// NETWORK 5
//   TCP_clear_error: <<<<<<<<<<<<<<<<<<<<<<<<<<<<<clear error>>>>>>>>>>>>>>>>>>>>>>>>>>>>>>>>>
//   axisdata[1].Axis_Error: A-0-0021.09 -RD- Axis reports error
//   axisdata[2].Axis_Error: A-0-0021.09 -RD- Axis reports error
//   axisdata[3].Axis_Error: A-0-0021.09 -RD- Axis reports error
//   FP_C_0_1030: Command: Clear all control errors
//   drive1: Real axis "Drive1" with axis number 1
// label: (*clear error*)
FB_clear_error_TCP(
    Execute := TCP_clear_error AND (axisdata[1].Axis_Error OR axisdata[2].Axis_Error OR axisdata[3].Axis_Error),
    ParameterNumber := FP_C_0_1030,
    Value := 3,
    Axis := drive1); // MB_WriteParameter
TCP_clear_done := FB_clear_error_TCP.Done;

// NETWORK 6
//   TCP_clear_error: <<<<<<<<<<<<<<<<<<<<<<<<<<<<<clear error>>>>>>>>>>>>>>>>>>>>>>>>>>>>>>>>>
//   b_enable_az_1: the enable of drive 1
//   b_enable_az_2: the enable of drive 2
//   b_enable_el_3: the enable of drive 3
// label: (*enable every driver under remote command*)
fb_rtrig_en_TCP(CLK := b_scc_enable_on AND TCP_clear_error); // R_TRIG
b_enable_az_1 S= fb_rtrig_en_TCP.Q;
b_enable_az_2 S= fb_rtrig_en_TCP.Q;
b_enable_el_3 S= fb_rtrig_en_TCP.Q;

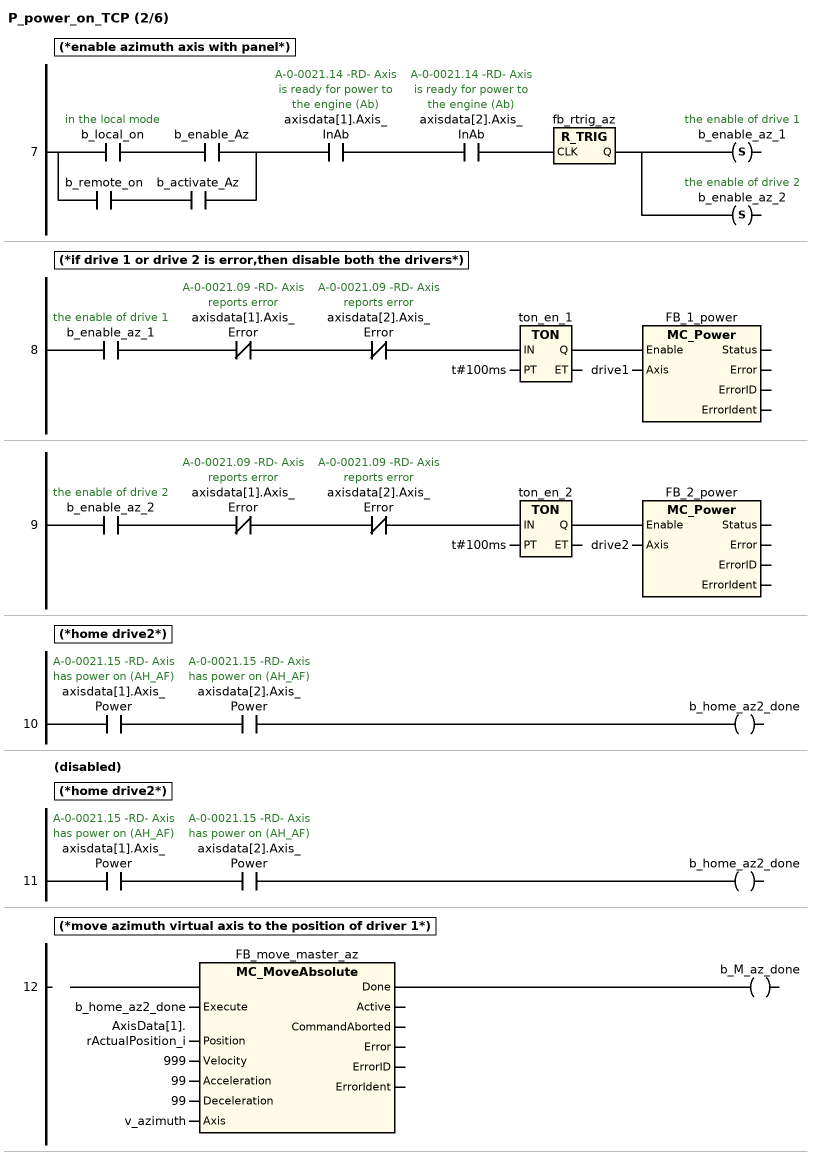
// NETWORK 7
//   b_local_on: in the local mode
//   axisdata[1].Axis_InAb: A-0-0021.14 -RD- Axis is ready for power to the engine (Ab)
//   axisdata[2].Axis_InAb: A-0-0021.14 -RD- Axis is ready for power to the engine (Ab)
//   b_enable_az_1: the enable of drive 1
//   b_enable_az_2: the enable of drive 2
// label: (*enable azimuth axis with panel*)
fb_rtrig_az(CLK := (b_local_on AND b_enable_Az OR b_remote_on AND b_activate_Az) AND axisdata[1].Axis_InAb AND axisdata[2].Axis_InAb); // R_TRIG
b_enable_az_1 S= fb_rtrig_az.Q;
b_enable_az_2 S= fb_rtrig_az.Q;

// NETWORK 8
//   FB_1_power: MC_Power function block controls the power connection (power on or off)
//   ton_en_1: <<<<<<<The function block Timer On Delay implements a turn-on delay>>>>>>
//   b_enable_az_1: the enable of drive 1
//   axisdata[1].Axis_Error: A-0-0021.09 -RD- Axis reports error
//   axisdata[2].Axis_Error: A-0-0021.09 -RD- Axis reports error
//   drive1: Real axis "Drive1" with axis number 1
// label: (*if drive 1 or drive 2 is error,then disable both the drivers*)
ton_en_1(IN := b_enable_az_1 AND NOT axisdata[1].Axis_Error AND NOT axisdata[2].Axis_Error, PT := t#100ms); // TON
FB_1_power(Enable := ton_en_1.Q, Axis := drive1); // MC_Power

// NETWORK 9
//   b_enable_az_2: the enable of drive 2
//   axisdata[1].Axis_Error: A-0-0021.09 -RD- Axis reports error
//   axisdata[2].Axis_Error: A-0-0021.09 -RD- Axis reports error
//   drive2: Real axis "Drive2" with axis number 2
ton_en_2(IN := b_enable_az_2 AND NOT axisdata[1].Axis_Error AND NOT axisdata[2].Axis_Error, PT := t#100ms); // TON
FB_2_power(Enable := ton_en_2.Q, Axis := drive2); // MC_Power

// NETWORK 10
//   axisdata[1].Axis_Power: A-0-0021.15 -RD- Axis has power on (AH_AF)
//   axisdata[2].Axis_Power: A-0-0021.15 -RD- Axis has power on (AH_AF)
// label: (*home drive2*)
b_home_az2_done := axisdata[1].Axis_Power AND axisdata[2].Axis_Power;

// NETWORK 11 (disabled)
//   axisdata[1].Axis_Power: A-0-0021.15 -RD- Axis has power on (AH_AF)
//   axisdata[2].Axis_Power: A-0-0021.15 -RD- Axis has power on (AH_AF)
// label: (*home drive2*)
// b_home_az2_done := axisdata[1].Axis_Power AND axisdata[2].Axis_Power;

// NETWORK 12
//   FB_move_master_az: "MC_MoveAbsolute" is used to move the drive to a preset absolute position.
//   AxisData[1].rActualPosition_i: A-0-0100 -RD- Actual position
//   v_azimuth: Virtual axis "v_azimuth" with axis number 7
// label: (*move azimuth virtual axis to the position of driver 1*)
FB_move_master_az(
    Execute := b_home_az2_done,
    Position := AxisData[1].rActualPosition_i,
    Velocity := 999,
    Acceleration := 99,
    Deceleration := 99,
    Axis := v_azimuth); // MC_MoveAbsolute
b_M_az_done := FB_move_master_az.Done;

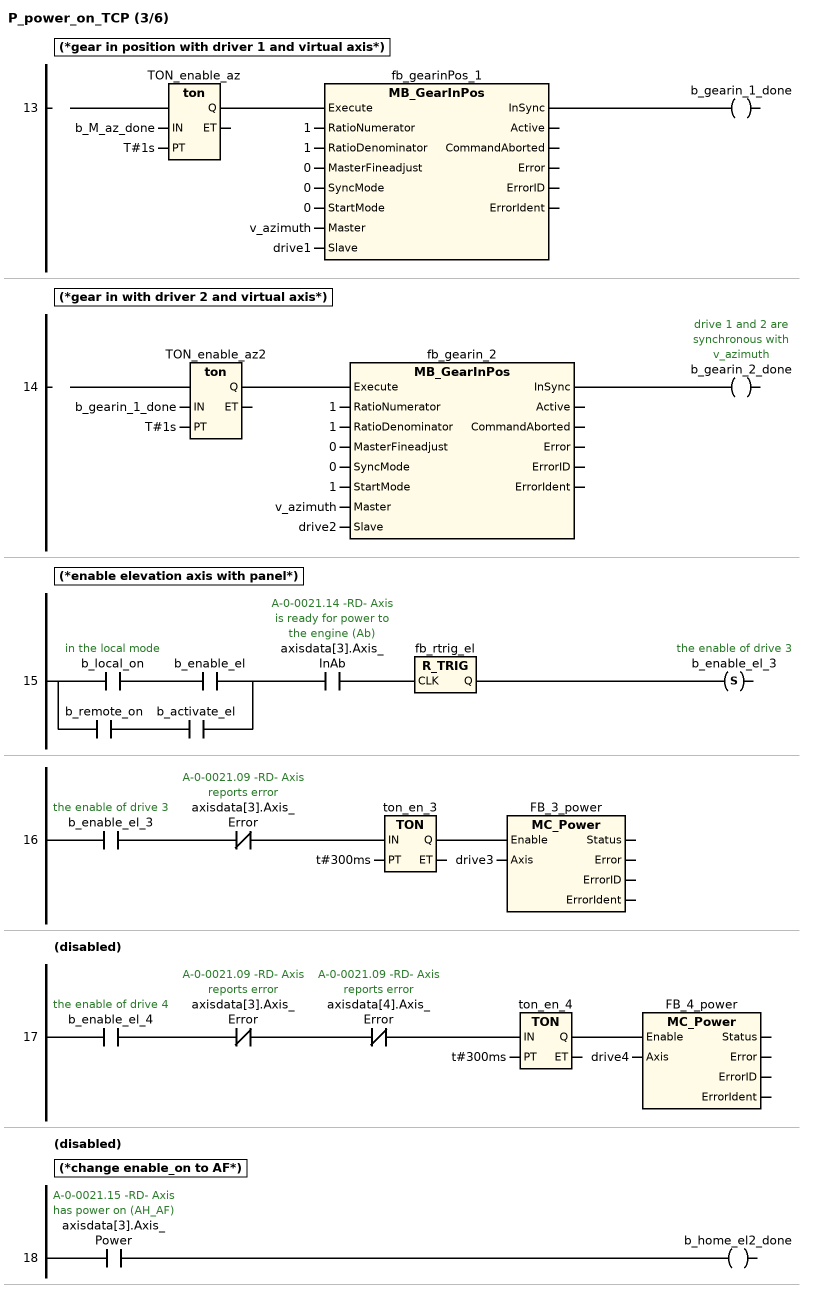
// NETWORK 13
//   fb_gearinPos_1: With "MB_GearInPos",it is possible to realize a motion of the slave axis which is phase synchronous to the master axis
//   v_azimuth: Virtual axis "v_azimuth" with axis number 7
//   drive1: Real axis "Drive1" with axis number 1
// label: (*gear in position with driver 1 and virtual axis*)
TON_enable_az(IN := b_M_az_done, PT := T#1s); // ton
fb_gearinPos_1(
    Execute := TON_enable_az.Q,
    RatioNumerator := 1,
    RatioDenominator := 1,
    MasterFineadjust := 0,
    SyncMode := 0,
    StartMode := 0,
    Master := v_azimuth,
    Slave := drive1); // MB_GearInPos
b_gearin_1_done := fb_gearinPos_1.InSync;

// NETWORK 14
//   v_azimuth: Virtual axis "v_azimuth" with axis number 7
//   drive2: Real axis "Drive2" with axis number 2
//   b_gearin_2_done: drive 1 and 2 are synchronous with v_azimuth
// label: (*gear in with driver 2 and virtual axis*)
TON_enable_az2(IN := b_gearin_1_done, PT := T#1s); // ton
fb_gearin_2(
    Execute := TON_enable_az2.Q,
    RatioNumerator := 1,
    RatioDenominator := 1,
    MasterFineadjust := 0,
    SyncMode := 0,
    StartMode := 1,
    Master := v_azimuth,
    Slave := drive2); // MB_GearInPos
b_gearin_2_done := fb_gearin_2.InSync;

// NETWORK 15
//   b_local_on: in the local mode
//   axisdata[3].Axis_InAb: A-0-0021.14 -RD- Axis is ready for power to the engine (Ab)
//   b_enable_el_3: the enable of drive 3
// label: (*enable elevation axis with panel*)
fb_rtrig_el(CLK := (b_local_on AND b_enable_el OR b_remote_on AND b_activate_el) AND axisdata[3].Axis_InAb); // R_TRIG
b_enable_el_3 S= fb_rtrig_el.Q;

// NETWORK 16
//   b_enable_el_3: the enable of drive 3
//   axisdata[3].Axis_Error: A-0-0021.09 -RD- Axis reports error
//   drive3: Real axis "Drive3" with axis number 3
ton_en_3(IN := b_enable_el_3 AND NOT axisdata[3].Axis_Error, PT := t#300ms); // TON
FB_3_power(Enable := ton_en_3.Q, Axis := drive3); // MC_Power

// NETWORK 17 (disabled)
//   b_enable_el_4: the enable of drive 4
//   axisdata[3].Axis_Error: A-0-0021.09 -RD- Axis reports error
//   axisdata[4].Axis_Error: A-0-0021.09 -RD- Axis reports error
//   drive4: Real axis "Drive4" with axis number 4
// ton_en_4(IN := b_enable_el_4 AND NOT axisdata[3].Axis_Error AND NOT axisdata[4].Axis_Error, PT := t#300ms); // TON
// FB_4_power(Enable := ton_en_4.Q, Axis := drive4); // MC_Power

// NETWORK 18 (disabled)
//   axisdata[3].Axis_Power: A-0-0021.15 -RD- Axis has power on (AH_AF)
// label: (*change enable_on to AF*)
// b_home_el2_done := axisdata[3].Axis_Power;

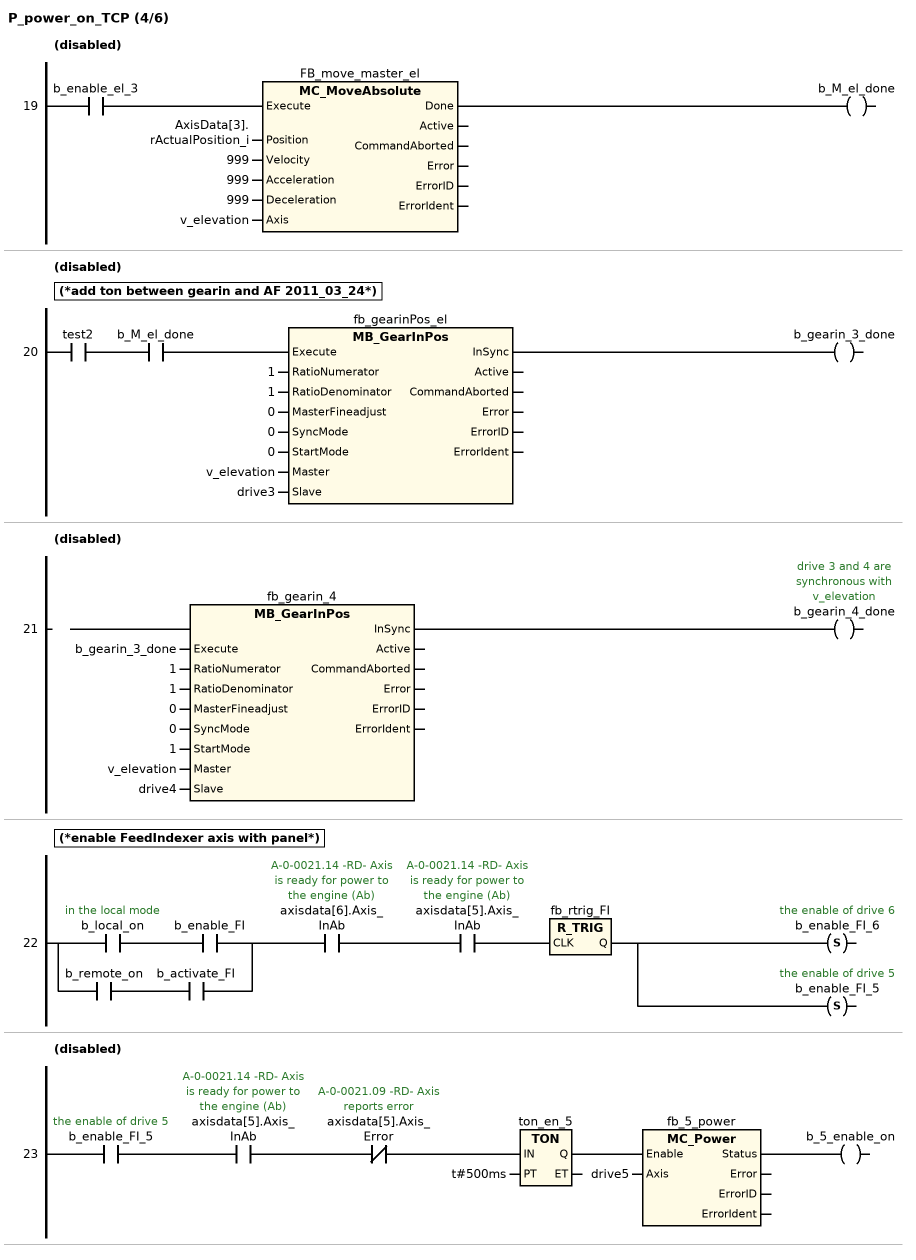
// NETWORK 19 (disabled)
//   AxisData[3].rActualPosition_i: A-0-0100 -RD- Actual position
//   v_elevation: Virtual axis "v_elevation" with axis number 8
// FB_move_master_el(
//     Execute := b_enable_el_3,
//     Position := AxisData[3].rActualPosition_i,
//     Velocity := 999,
//     Acceleration := 999,
//     Deceleration := 999,
//     Axis := v_elevation); // MC_MoveAbsolute
// b_M_el_done := FB_move_master_el.Done;

// NETWORK 20 (disabled)
//   fb_gearinPos_el: add 2011 06 09 to delete 1sec delay
//   v_elevation: Virtual axis "v_elevation" with axis number 8
//   drive3: Real axis "Drive3" with axis number 3
// label: (*add ton between gearin and AF 2011_03_24*)
// fb_gearinPos_el(
//     Execute := test2 AND b_M_el_done,
//     RatioNumerator := 1,
//     RatioDenominator := 1,
//     MasterFineadjust := 0,
//     SyncMode := 0,
//     StartMode := 0,
//     Master := v_elevation,
//     Slave := drive3); // MB_GearInPos
// b_gearin_3_done := fb_gearinPos_el.InSync;

// NETWORK 21 (disabled)
//   v_elevation: Virtual axis "v_elevation" with axis number 8
//   drive4: Real axis "Drive4" with axis number 4
//   b_gearin_4_done: drive 3 and 4 are synchronous with v_elevation
// fb_gearin_4(
//     Execute := b_gearin_3_done,
//     RatioNumerator := 1,
//     RatioDenominator := 1,
//     MasterFineadjust := 0,
//     SyncMode := 0,
//     StartMode := 1,
//     Master := v_elevation,
//     Slave := drive4); // MB_GearInPos
// b_gearin_4_done := fb_gearin_4.InSync;

// NETWORK 22
//   b_local_on: in the local mode
//   axisdata[6].Axis_InAb: A-0-0021.14 -RD- Axis is ready for power to the engine (Ab)
//   axisdata[5].Axis_InAb: A-0-0021.14 -RD- Axis is ready for power to the engine (Ab)
//   b_enable_FI_6: the enable of drive 6
//   b_enable_FI_5: the enable of drive 5
// label: (*enable FeedIndexer axis with panel*)
fb_rtrig_FI(CLK := (b_local_on AND b_enable_FI OR b_remote_on AND b_activate_FI) AND axisdata[6].Axis_InAb AND axisdata[5].Axis_InAb); // R_TRIG
b_enable_FI_6 S= fb_rtrig_FI.Q;
b_enable_FI_5 S= fb_rtrig_FI.Q;

// NETWORK 23 (disabled)
//   b_enable_FI_5: the enable of drive 5
//   axisdata[5].Axis_InAb: A-0-0021.14 -RD- Axis is ready for power to the engine (Ab)
//   axisdata[5].Axis_Error: A-0-0021.09 -RD- Axis reports error
//   drive5: Real axis "Drive5" with axis number 5
// ton_en_5(IN := b_enable_FI_5 AND axisdata[5].Axis_InAb AND NOT axisdata[5].Axis_Error, PT := t#500ms); // TON
// fb_5_power(Enable := ton_en_5.Q, Axis := drive5); // MC_Power
// b_5_enable_on := fb_5_power.Status;

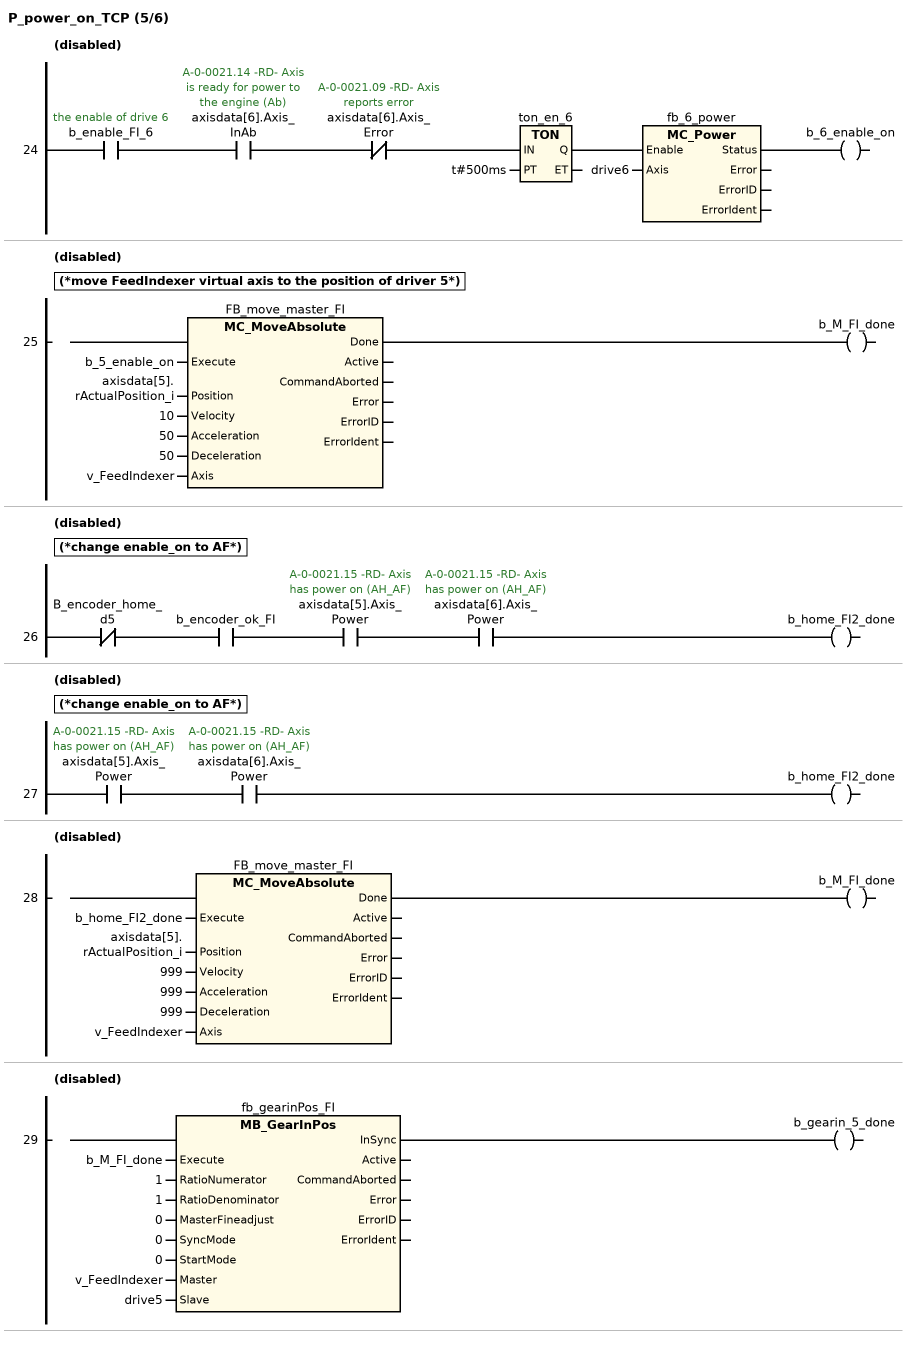
// NETWORK 24 (disabled)
//   b_enable_FI_6: the enable of drive 6
//   axisdata[6].Axis_InAb: A-0-0021.14 -RD- Axis is ready for power to the engine (Ab)
//   axisdata[6].Axis_Error: A-0-0021.09 -RD- Axis reports error
//   drive6: Real axis "Drive6" with axis number 6
// ton_en_6(IN := b_enable_FI_6 AND axisdata[6].Axis_InAb AND NOT axisdata[6].Axis_Error, PT := t#500ms); // TON
// fb_6_power(Enable := ton_en_6.Q, Axis := drive6); // MC_Power
// b_6_enable_on := fb_6_power.Status;

// NETWORK 25 (disabled)
//   axisdata[5].rActualPosition_i: A-0-0100 -RD- Actual position
//   v_FeedIndexer: Virtual axis "v_polarization" with axis number 9
// label: (*move FeedIndexer virtual axis to the position of driver 5*)
// FB_move_master_FI(
//     Execute := b_5_enable_on,
//     Position := axisdata[5].rActualPosition_i,
//     Velocity := 10,
//     Acceleration := 50,
//     Deceleration := 50,
//     Axis := v_FeedIndexer); // MC_MoveAbsolute
// b_M_FI_done := FB_move_master_FI.Done;

// NETWORK 26 (disabled)
//   axisdata[5].Axis_Power: A-0-0021.15 -RD- Axis has power on (AH_AF)
//   axisdata[6].Axis_Power: A-0-0021.15 -RD- Axis has power on (AH_AF)
// label: (*change enable_on to AF*)
// b_home_FI2_done := NOT B_encoder_home_d5 AND b_encoder_ok_FI AND axisdata[5].Axis_Power AND axisdata[6].Axis_Power;

// NETWORK 27 (disabled)
//   axisdata[5].Axis_Power: A-0-0021.15 -RD- Axis has power on (AH_AF)
//   axisdata[6].Axis_Power: A-0-0021.15 -RD- Axis has power on (AH_AF)
// label: (*change enable_on to AF*)
// b_home_FI2_done := axisdata[5].Axis_Power AND axisdata[6].Axis_Power;

// NETWORK 28 (disabled)
//   axisdata[5].rActualPosition_i: A-0-0100 -RD- Actual position
//   v_FeedIndexer: Virtual axis "v_polarization" with axis number 9
// FB_move_master_FI(
//     Execute := b_home_FI2_done,
//     Position := axisdata[5].rActualPosition_i,
//     Velocity := 999,
//     Acceleration := 999,
//     Deceleration := 999,
//     Axis := v_FeedIndexer); // MC_MoveAbsolute
// b_M_FI_done := FB_move_master_FI.Done;

// NETWORK 29 (disabled)
//   v_FeedIndexer: Virtual axis "v_polarization" with axis number 9
//   drive5: Real axis "Drive5" with axis number 5
// fb_gearinPos_FI(
//     Execute := b_M_FI_done,
//     RatioNumerator := 1,
//     RatioDenominator := 1,
//     MasterFineadjust := 0,
//     SyncMode := 0,
//     StartMode := 0,
//     Master := v_FeedIndexer,
//     Slave := drive5); // MB_GearInPos
// b_gearin_5_done := fb_gearinPos_FI.InSync;

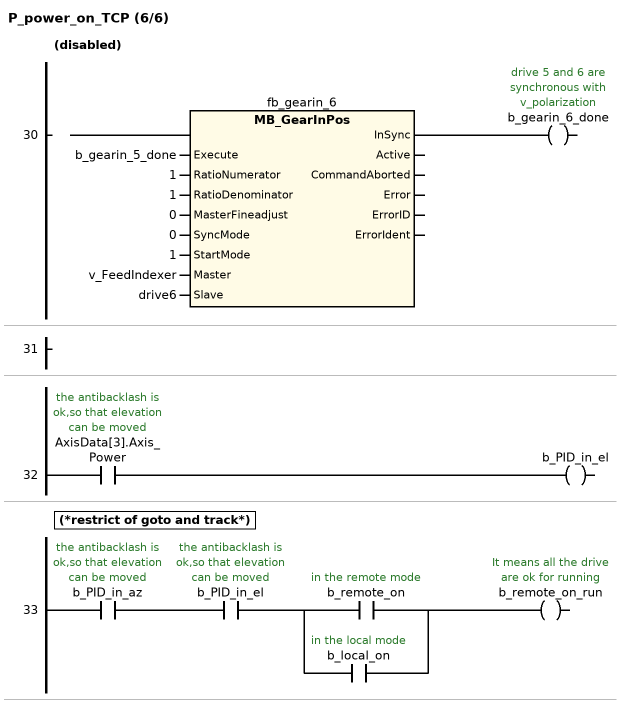
// NETWORK 30 (disabled)
//   v_FeedIndexer: Virtual axis "v_polarization" with axis number 9
//   drive6: Real axis "Drive6" with axis number 6
//   b_gearin_6_done: drive 5 and 6 are synchronous with v_polarization
// fb_gearin_6(
//     Execute := b_gearin_5_done,
//     RatioNumerator := 1,
//     RatioDenominator := 1,
//     MasterFineadjust := 0,
//     SyncMode := 0,
//     StartMode := 1,
//     Master := v_FeedIndexer,
//     Slave := drive6); // MB_GearInPos
// b_gearin_6_done := fb_gearin_6.InSync;

// NETWORK 31

// NETWORK 32
//   AxisData[3].Axis_Power: the antibacklash is ok,so that elevation can be moved
b_PID_in_el := AxisData[3].Axis_Power;

// NETWORK 33
//   b_PID_in_az: the antibacklash is ok,so that elevation can be moved
//   b_PID_in_el: the antibacklash is ok,so that elevation can be moved
//   b_remote_on: in the remote mode
//   b_local_on: in the local mode
//   b_remote_on_run: It means all the drive are ok for running
// label: (*restrict of goto and track*)
b_remote_on_run := b_PID_in_az AND b_PID_in_el AND (b_remote_on OR b_local_on);

END_PROGRAM

// IndraMotionMlc1/Application/POUs/Panel Function/P_remote_local
(*This program is built for switch the mode between local,remote and off.
In the local mode,the antenna can be controled only by the button on the
panelbox;In the remote mode,the antenna can be controled only by the command
that come from the ACU;In the off mode,all the motion will be stopped.
And every time the switch is off,there is a clear_error action*)
PROGRAM P_remote_local
VAR
(*clear all error when the switch is off*)
	FB_clear_all_error: MB_WriteParameter;
	b_clear_error: BOOL;
	b_clear_all_error: BOOL;
	b_clear_done: BOOL;
	rtrig_clear_error: R_TRIG;
	rtrig_reset_clear: R_TRIG;
	
END_VAR


IF b_HHP_connected THEN
	b_remote_on:=FALSE;
	b_local_on:=TRUE;
	CommandArbiter.Status.DscCmdAuthority:= HHP; // Needsome code to change it to No Auth when HHP is dosconnected. 
ELSE
	b_remote_on:=TRUE;
	b_local_on:=FALSE;
END_IF

IF b_local_on OR b_remote_on THEN
	b_clear_error:=FALSE;
END_IF;
(*when the switch is off,reset some command and stop all the motion*)
IF b_remote_on =FALSE AND b_local_on=FALSE THEN
	b_power_Az:=FALSE;
	b_power_el:=FALSE;
	b_power_FI:=FALSE;
	b_stow_pin_deploy:=FALSE;
	b_stow_pin_retract:=FALSE;
	b_scc_enable_on:=FALSE;
	b_scc_enable_off:=FALSE;
	b_scc_stow:=FALSE;
	b_track_on:=FALSE;
	b_clear_error:=TRUE;
	b_scc_goto:=FALSE;
	b_scc_goto_az:=FALSE;
	b_scc_goto_el:=FALSE;
	b_scc_goto_FI:=FALSE;
	b_scc_vel:=FALSE;
END_IF;
(*transfer the sub-program A_clear_error to clear all the error*)
P_remote_local.A_clear_error();

ACTION A_clear_error:
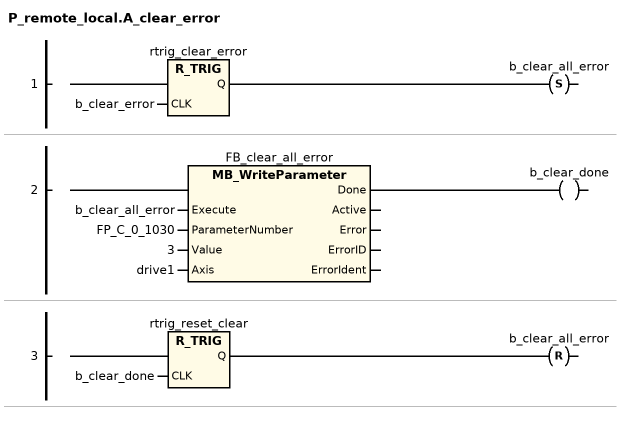
// NETWORK 1
rtrig_clear_error(CLK := b_clear_error); // R_TRIG
b_clear_all_error S= rtrig_clear_error.Q;

// NETWORK 2
FB_clear_all_error(Execute := b_clear_all_error, ParameterNumber := FP_C_0_1030, Value := 3, Axis := drive1); // MB_WriteParameter
b_clear_done := FB_clear_all_error.Done;

// NETWORK 3
rtrig_reset_clear(CLK := b_clear_done); // R_TRIG
b_clear_all_error R= rtrig_reset_clear.Q;
END_ACTION

END_PROGRAM

// IndraMotionMlc1/Application/POUs/Motion/P_power_on_Sim
(*the program is built for power on the 3 axis under the contol of remote or local.
the elevation axis is the similar with the azimuth*)
PROGRAM P_power_on_Sim
VAR
(*<<<<<<<<definition of r_trig for detecting a rising edge>>>>>>>>>>>>>>*)
	fb_rtrig_p1: R_TRIG;
	fb_rtrig_p3: R_TRIG;
	fb_rtrig_p5: R_TRIG;
	fb_rtrig_az: R_TRIG;
	fb_rtrig_el: R_TRIG;
	fb_rtrig_FI: R_TRIG;
	fb_rtrig_en_remote: R_TRIG;
	fb_rtrig_en_TCP: R_TRIG;
(*<<<<<<<The function block Timer On Delay implements a turn-on delay>>>>>>*)
	ton_en_1: TON;
	ton_en_2: TON;
	ton_en_3: TON;
	ton_en_4: TON;
	ton_en_5: TON;
	ton_en_6: TON;
(*MC_Power function block controls the power connection (power on or off)*)
	FB_1_power: MC_Power;
	FB_2_power: MC_Power;
	FB_3_power: MC_Power;
	FB_4_power: MC_Power;
	FB_5_power: MC_Power;
	FB_6_power: MC_Power;
	b_1_enable_on: BOOL;
	b_2_enable_on: BOOL;
	b_3_enable_on: BOOL;
	b_4_enable_on: BOOL;
	b_5_enable_on: BOOL;
	b_6_enable_on: BOOL;
(*With "MB_GearInPos",it is possible to realize a motion of the slave axis which is phase synchronous to the master axis*)
	fb_gearinPos_1: MB_GearInPos;
	fb_gearin_2: MB_GearInPos;
	fb_gearinPos_3: MB_GearInPos;
	fb_gearin_4: MB_GearInPos;
	fb_gearinPos_5: MB_GearInPos;
	fb_gearin_6: MB_GearInPos;
	b_gearin_1_done: BOOL;
	
	b_gearin_5_done:BOOL;
(*"MC_MoveAbsolute" is used to move the drive to a preset absolute position.*)
	FB_move_master_az: MC_MoveAbsolute;
	FB_move_master_el: MC_MoveAbsolute;
	FB_move_master_FI: MC_MoveAbsolute;
	b_M_az_done: BOOL;
	b_M_el_done: BOOL;
	b_M_FI_done: BOOL;
(*MB_Home function block controls axes with incremental encoder when executing the "search home" sequence*)
	fb_home_az2: MB_Home;
	fb_home_el2: MB_Home;
	fb_home_FI2: MB_Home;
	b_home_az2_done: BOOL;
	b_home_el2_done: BOOL;
	b_home_FI2_done: BOOL;
(*<<<<<<<<<<<<<<<<<<<<<<<<<<<<<clear error>>>>>>>>>>>>>>>>>>>>>>>>>>>>>>>>>*)
	TCP_clear_error: BOOL;
	FB_clear_error_TCP: MB_WriteParameter;
	TCP_clear_done: BOOL;
(*add 2011 06 09 to delete 1sec delay*)
	fb_gearinPos_el: MB_GearInPos;
	b_gearin_el_done: BOOL;
	fb_gearout_el: MC_GearOut;
	rtrig_set_gearin_3: R_TRIG;
	b_gearin_3: BOOL;
	rtrig_reset_gearin_3: F_TRIG;
	ton_clear_on: TON;
	fb_gearinPos_FI: MB_GearInPos;
	test_111: BOOL;
	ssss: BOOL;
	test1: BOOL;
	test2: BOOL;
	test3: BOOL;
	TON_enable_az: ton;
	TON_enable_az2: ton;
	fb_gearPos_2: MB_GearInPos;
	TON_enable_el: ton;
	b_M_el_done_1: BOOL;
	R_TRIG_0: R_TRIG;
END_VAR

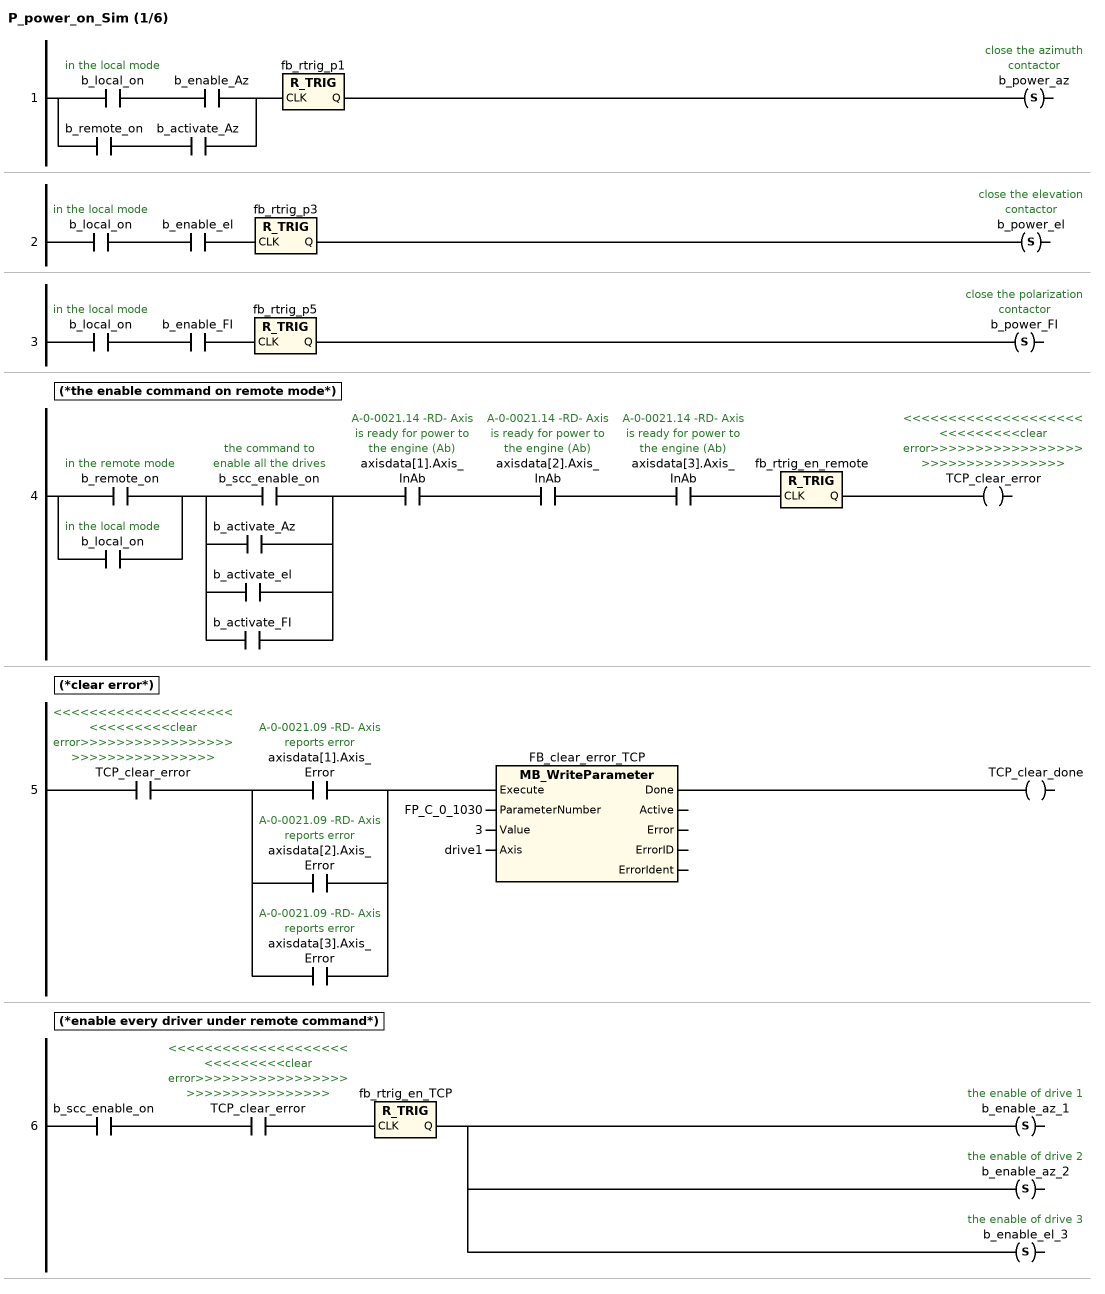
// NETWORK 1
//   fb_rtrig_p1: <<<<<<<<definition of r_trig for detecting a rising edge>>>>>>>>>>>>>>
//   b_local_on: in the local mode
//   b_power_az: close the azimuth contactor
fb_rtrig_p1(CLK := b_local_on AND b_enable_Az OR b_remote_on AND b_activate_Az); // R_TRIG
b_power_az S= fb_rtrig_p1.Q;

// NETWORK 2
//   b_local_on: in the local mode
//   b_power_el: close the elevation contactor
fb_rtrig_p3(CLK := b_local_on AND b_enable_el); // R_TRIG
b_power_el S= fb_rtrig_p3.Q;

// NETWORK 3
//   b_local_on: in the local mode
//   b_power_FI: close the polarization contactor
fb_rtrig_p5(CLK := b_local_on AND b_enable_FI); // R_TRIG
b_power_FI S= fb_rtrig_p5.Q;

// NETWORK 4
//   b_remote_on: in the remote mode
//   b_local_on: in the local mode
//   b_scc_enable_on: the command to enable all the drives
//   axisdata[1].Axis_InAb: A-0-0021.14 -RD- Axis is ready for power to the engine (Ab)
//   axisdata[2].Axis_InAb: A-0-0021.14 -RD- Axis is ready for power to the engine (Ab)
//   axisdata[3].Axis_InAb: A-0-0021.14 -RD- Axis is ready for power to the engine (Ab)
//   TCP_clear_error: <<<<<<<<<<<<<<<<<<<<<<<<<<<<<clear error>>>>>>>>>>>>>>>>>>>>>>>>>>>>>>>>>
// label: (*the enable command on remote mode*)
fb_rtrig_en_remote(CLK := (b_remote_on OR b_local_on) AND (b_scc_enable_on OR b_activate_Az OR b_activate_el OR b_activate_FI) AND axisdata[1].Axis_InAb AND axisdata[2].Axis_InAb AND axisdata[3].Axis_InAb); // R_TRIG
TCP_clear_error := fb_rtrig_en_remote.Q;

// NETWORK 5
//   TCP_clear_error: <<<<<<<<<<<<<<<<<<<<<<<<<<<<<clear error>>>>>>>>>>>>>>>>>>>>>>>>>>>>>>>>>
//   axisdata[1].Axis_Error: A-0-0021.09 -RD- Axis reports error
//   axisdata[2].Axis_Error: A-0-0021.09 -RD- Axis reports error
//   axisdata[3].Axis_Error: A-0-0021.09 -RD- Axis reports error
//   FP_C_0_1030: Command: Clear all control errors
//   drive1: Real axis "Drive1" with axis number 1
// label: (*clear error*)
FB_clear_error_TCP(
    Execute := TCP_clear_error AND (axisdata[1].Axis_Error OR axisdata[2].Axis_Error OR axisdata[3].Axis_Error),
    ParameterNumber := FP_C_0_1030,
    Value := 3,
    Axis := drive1); // MB_WriteParameter
TCP_clear_done := FB_clear_error_TCP.Done;

// NETWORK 6
//   TCP_clear_error: <<<<<<<<<<<<<<<<<<<<<<<<<<<<<clear error>>>>>>>>>>>>>>>>>>>>>>>>>>>>>>>>>
//   b_enable_az_1: the enable of drive 1
//   b_enable_az_2: the enable of drive 2
//   b_enable_el_3: the enable of drive 3
// label: (*enable every driver under remote command*)
fb_rtrig_en_TCP(CLK := b_scc_enable_on AND TCP_clear_error); // R_TRIG
b_enable_az_1 S= fb_rtrig_en_TCP.Q;
b_enable_az_2 S= fb_rtrig_en_TCP.Q;
b_enable_el_3 S= fb_rtrig_en_TCP.Q;

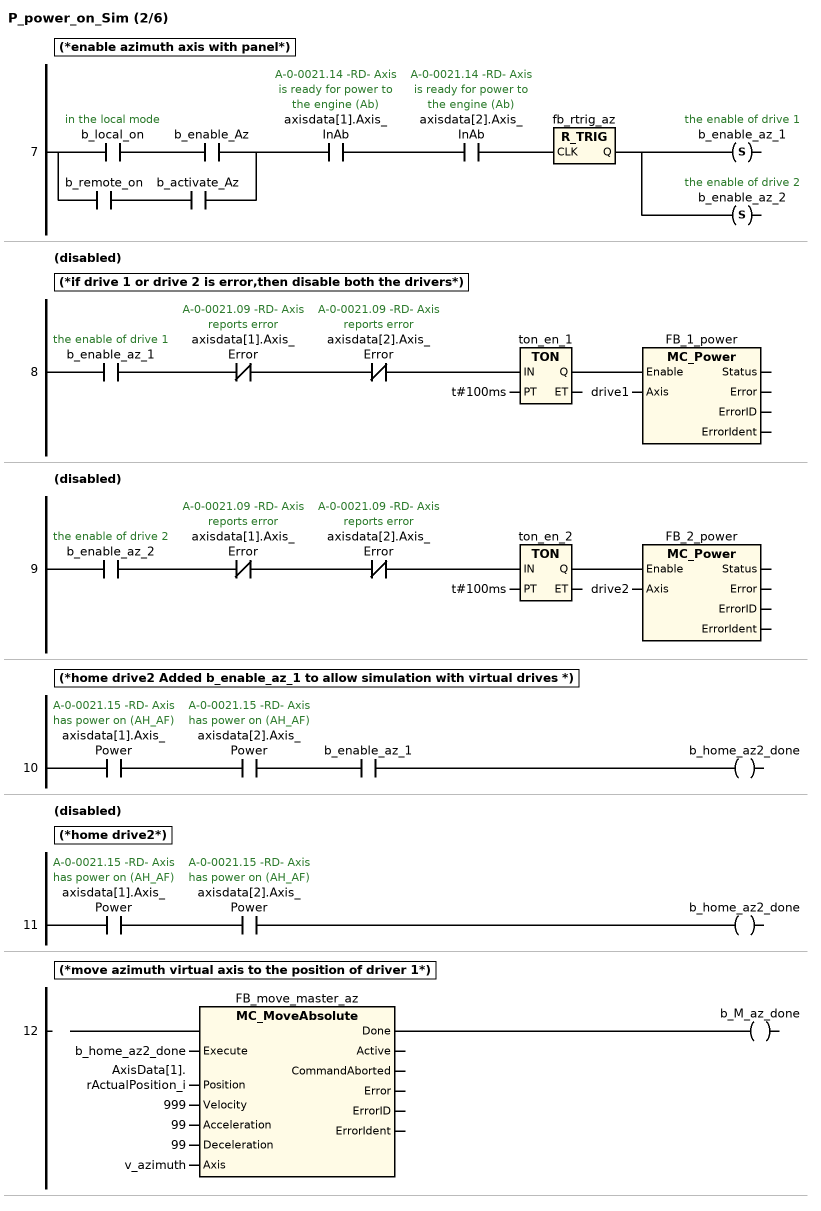
// NETWORK 7
//   b_local_on: in the local mode
//   axisdata[1].Axis_InAb: A-0-0021.14 -RD- Axis is ready for power to the engine (Ab)
//   axisdata[2].Axis_InAb: A-0-0021.14 -RD- Axis is ready for power to the engine (Ab)
//   b_enable_az_1: the enable of drive 1
//   b_enable_az_2: the enable of drive 2
// label: (*enable azimuth axis with panel*)
fb_rtrig_az(CLK := (b_local_on AND b_enable_Az OR b_remote_on AND b_activate_Az) AND axisdata[1].Axis_InAb AND axisdata[2].Axis_InAb); // R_TRIG
b_enable_az_1 S= fb_rtrig_az.Q;
b_enable_az_2 S= fb_rtrig_az.Q;

// NETWORK 8 (disabled)
//   FB_1_power: MC_Power function block controls the power connection (power on or off)
//   ton_en_1: <<<<<<<The function block Timer On Delay implements a turn-on delay>>>>>>
//   b_enable_az_1: the enable of drive 1
//   axisdata[1].Axis_Error: A-0-0021.09 -RD- Axis reports error
//   axisdata[2].Axis_Error: A-0-0021.09 -RD- Axis reports error
//   drive1: Real axis "Drive1" with axis number 1
// label: (*if drive 1 or drive 2 is error,then disable both the drivers*)
// ton_en_1(IN := b_enable_az_1 AND NOT axisdata[1].Axis_Error AND NOT axisdata[2].Axis_Error, PT := t#100ms); // TON
// FB_1_power(Enable := ton_en_1.Q, Axis := drive1); // MC_Power

// NETWORK 9 (disabled)
//   b_enable_az_2: the enable of drive 2
//   axisdata[1].Axis_Error: A-0-0021.09 -RD- Axis reports error
//   axisdata[2].Axis_Error: A-0-0021.09 -RD- Axis reports error
//   drive2: Real axis "Drive2" with axis number 2
// ton_en_2(IN := b_enable_az_2 AND NOT axisdata[1].Axis_Error AND NOT axisdata[2].Axis_Error, PT := t#100ms); // TON
// FB_2_power(Enable := ton_en_2.Q, Axis := drive2); // MC_Power

// NETWORK 10
//   axisdata[1].Axis_Power: A-0-0021.15 -RD- Axis has power on (AH_AF)
//   axisdata[2].Axis_Power: A-0-0021.15 -RD- Axis has power on (AH_AF)
// label: (*home drive2 Added b_enable_az_1 to allow simulation with virtual drives *)
b_home_az2_done := axisdata[1].Axis_Power AND axisdata[2].Axis_Power AND b_enable_az_1;

// NETWORK 11 (disabled)
//   axisdata[1].Axis_Power: A-0-0021.15 -RD- Axis has power on (AH_AF)
//   axisdata[2].Axis_Power: A-0-0021.15 -RD- Axis has power on (AH_AF)
// label: (*home drive2*)
// b_home_az2_done := axisdata[1].Axis_Power AND axisdata[2].Axis_Power;

// NETWORK 12
//   FB_move_master_az: "MC_MoveAbsolute" is used to move the drive to a preset absolute position.
//   AxisData[1].rActualPosition_i: A-0-0100 -RD- Actual position
//   v_azimuth: Virtual axis "v_azimuth" with axis number 7
// label: (*move azimuth virtual axis to the position of driver 1*)
FB_move_master_az(
    Execute := b_home_az2_done,
    Position := AxisData[1].rActualPosition_i,
    Velocity := 999,
    Acceleration := 99,
    Deceleration := 99,
    Axis := v_azimuth); // MC_MoveAbsolute
b_M_az_done := FB_move_master_az.Done;

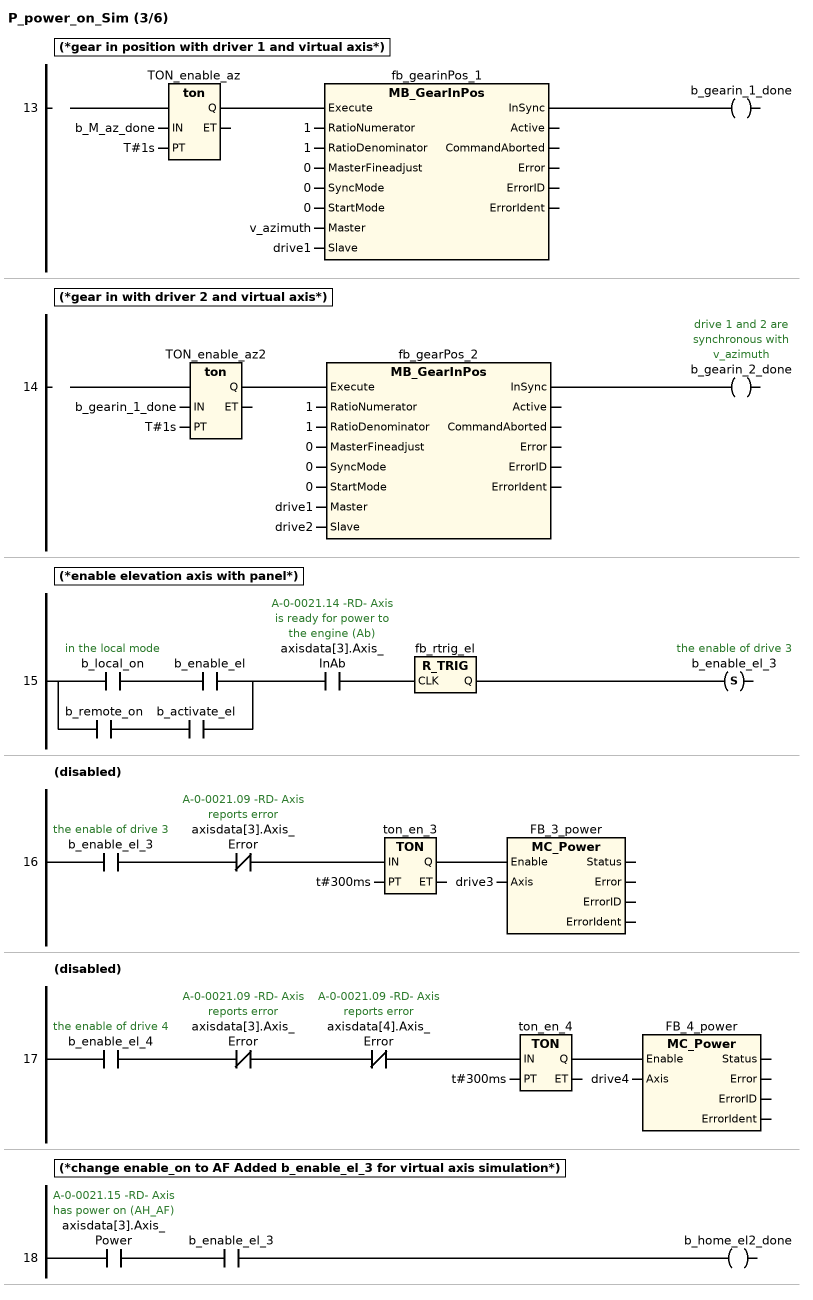
// NETWORK 13
//   fb_gearinPos_1: With "MB_GearInPos",it is possible to realize a motion of the slave axis which is phase synchronous to the master axis
//   v_azimuth: Virtual axis "v_azimuth" with axis number 7
//   drive1: Real axis "Drive1" with axis number 1
// label: (*gear in position with driver 1 and virtual axis*)
TON_enable_az(IN := b_M_az_done, PT := T#1s); // ton
fb_gearinPos_1(
    Execute := TON_enable_az.Q,
    RatioNumerator := 1,
    RatioDenominator := 1,
    MasterFineadjust := 0,
    SyncMode := 0,
    StartMode := 0,
    Master := v_azimuth,
    Slave := drive1); // MB_GearInPos
b_gearin_1_done := fb_gearinPos_1.InSync;

// NETWORK 14
//   drive1: Virtual axis "v_azimuth" with axis number 7
//   drive2: Real axis "Drive2" with axis number 2
//   b_gearin_2_done: drive 1 and 2 are synchronous with v_azimuth
// label: (*gear in with driver 2 and virtual axis*)
TON_enable_az2(IN := b_gearin_1_done, PT := T#1s); // ton
fb_gearPos_2(
    Execute := TON_enable_az2.Q,
    RatioNumerator := 1,
    RatioDenominator := 1,
    MasterFineadjust := 0,
    SyncMode := 0,
    StartMode := 0,
    Master := drive1,
    Slave := drive2); // MB_GearInPos
b_gearin_2_done := fb_gearPos_2.InSync;

// NETWORK 15
//   b_local_on: in the local mode
//   axisdata[3].Axis_InAb: A-0-0021.14 -RD- Axis is ready for power to the engine (Ab)
//   b_enable_el_3: the enable of drive 3
// label: (*enable elevation axis with panel*)
fb_rtrig_el(CLK := (b_local_on AND b_enable_el OR b_remote_on AND b_activate_el) AND axisdata[3].Axis_InAb); // R_TRIG
b_enable_el_3 S= fb_rtrig_el.Q;

// NETWORK 16 (disabled)
//   b_enable_el_3: the enable of drive 3
//   axisdata[3].Axis_Error: A-0-0021.09 -RD- Axis reports error
//   drive3: Real axis "Drive3" with axis number 3
// ton_en_3(IN := b_enable_el_3 AND NOT axisdata[3].Axis_Error, PT := t#300ms); // TON
// FB_3_power(Enable := ton_en_3.Q, Axis := drive3); // MC_Power

// NETWORK 17 (disabled)
//   b_enable_el_4: the enable of drive 4
//   axisdata[3].Axis_Error: A-0-0021.09 -RD- Axis reports error
//   axisdata[4].Axis_Error: A-0-0021.09 -RD- Axis reports error
//   drive4: Real axis "Drive4" with axis number 4
// ton_en_4(IN := b_enable_el_4 AND NOT axisdata[3].Axis_Error AND NOT axisdata[4].Axis_Error, PT := t#300ms); // TON
// FB_4_power(Enable := ton_en_4.Q, Axis := drive4); // MC_Power

// NETWORK 18
//   axisdata[3].Axis_Power: A-0-0021.15 -RD- Axis has power on (AH_AF)
// label: (*change enable_on to AF Added b_enable_el_3 for virtual axis simulation*)
b_home_el2_done := axisdata[3].Axis_Power AND b_enable_el_3;

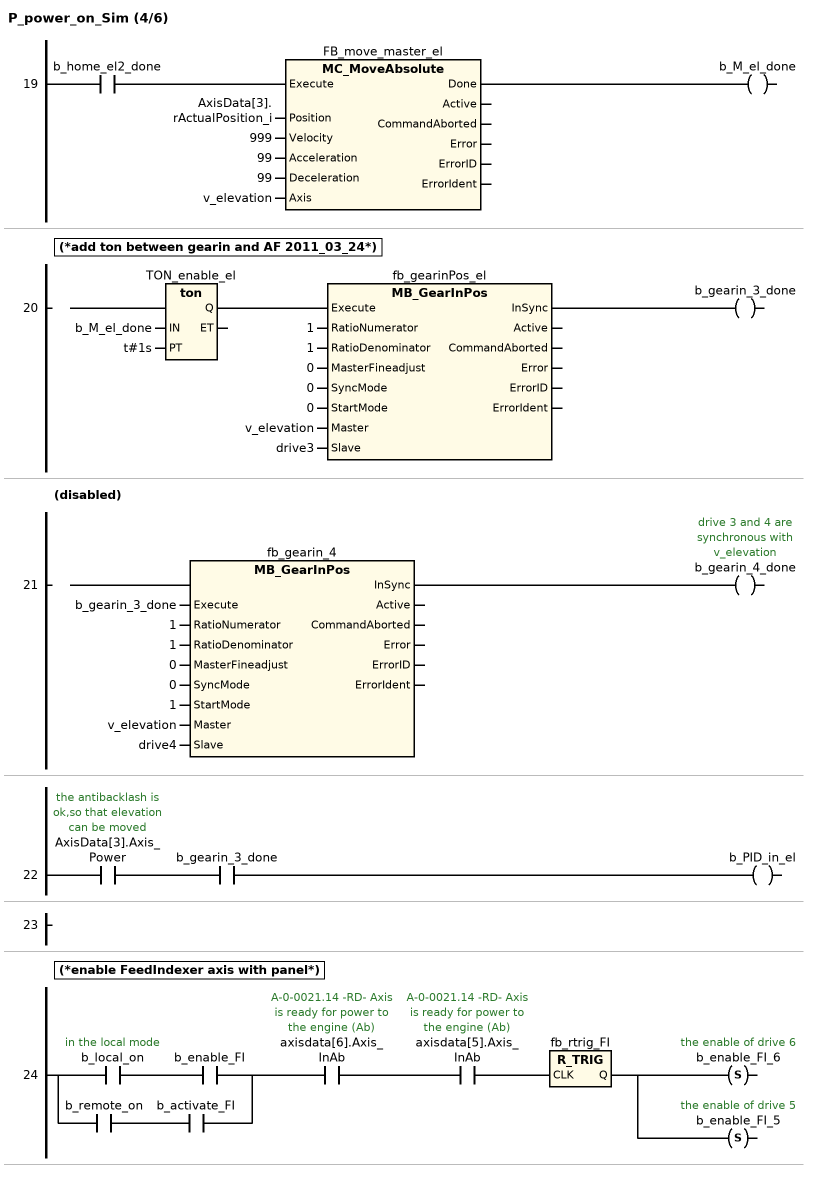
// NETWORK 19
//   AxisData[3].rActualPosition_i: A-0-0100 -RD- Actual position
//   v_elevation: Virtual axis "v_elevation" with axis number 8
FB_move_master_el(
    Execute := b_home_el2_done,
    Position := AxisData[3].rActualPosition_i,
    Velocity := 999,
    Acceleration := 99,
    Deceleration := 99,
    Axis := v_elevation); // MC_MoveAbsolute
b_M_el_done := FB_move_master_el.Done;

// NETWORK 20
//   fb_gearinPos_el: add 2011 06 09 to delete 1sec delay
//   v_elevation: Virtual axis "v_elevation" with axis number 8
//   drive3: Real axis "Drive3" with axis number 3
// label: (*add ton between gearin and AF 2011_03_24*)
TON_enable_el(IN := b_M_el_done, PT := t#1s); // ton
fb_gearinPos_el(
    Execute := TON_enable_el.Q,
    RatioNumerator := 1,
    RatioDenominator := 1,
    MasterFineadjust := 0,
    SyncMode := 0,
    StartMode := 0,
    Master := v_elevation,
    Slave := drive3); // MB_GearInPos
b_gearin_3_done := fb_gearinPos_el.InSync;

// NETWORK 21 (disabled)
//   v_elevation: Virtual axis "v_elevation" with axis number 8
//   drive4: Real axis "Drive4" with axis number 4
//   b_gearin_4_done: drive 3 and 4 are synchronous with v_elevation
// fb_gearin_4(
//     Execute := b_gearin_3_done,
//     RatioNumerator := 1,
//     RatioDenominator := 1,
//     MasterFineadjust := 0,
//     SyncMode := 0,
//     StartMode := 1,
//     Master := v_elevation,
//     Slave := drive4); // MB_GearInPos
// b_gearin_4_done := fb_gearin_4.InSync;

// NETWORK 22
//   AxisData[3].Axis_Power: the antibacklash is ok,so that elevation can be moved
b_PID_in_el := AxisData[3].Axis_Power AND b_gearin_3_done;

// NETWORK 23

// NETWORK 24
//   b_local_on: in the local mode
//   axisdata[6].Axis_InAb: A-0-0021.14 -RD- Axis is ready for power to the engine (Ab)
//   axisdata[5].Axis_InAb: A-0-0021.14 -RD- Axis is ready for power to the engine (Ab)
//   b_enable_FI_6: the enable of drive 6
//   b_enable_FI_5: the enable of drive 5
// label: (*enable FeedIndexer axis with panel*)
fb_rtrig_FI(CLK := (b_local_on AND b_enable_FI OR b_remote_on AND b_activate_FI) AND axisdata[6].Axis_InAb AND axisdata[5].Axis_InAb); // R_TRIG
b_enable_FI_6 S= fb_rtrig_FI.Q;
b_enable_FI_5 S= fb_rtrig_FI.Q;

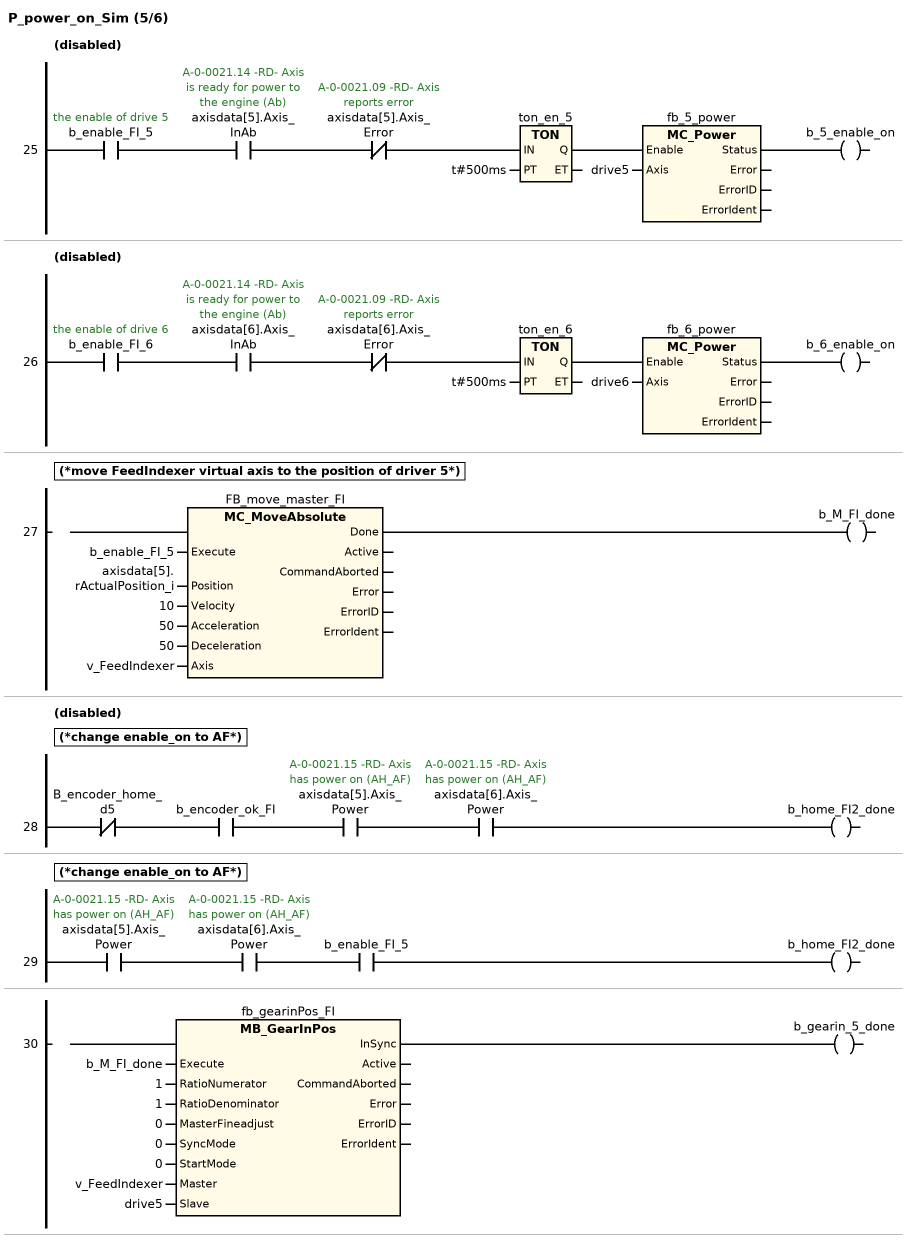
// NETWORK 25 (disabled)
//   b_enable_FI_5: the enable of drive 5
//   axisdata[5].Axis_InAb: A-0-0021.14 -RD- Axis is ready for power to the engine (Ab)
//   axisdata[5].Axis_Error: A-0-0021.09 -RD- Axis reports error
//   drive5: Real axis "Drive5" with axis number 5
// ton_en_5(IN := b_enable_FI_5 AND axisdata[5].Axis_InAb AND NOT axisdata[5].Axis_Error, PT := t#500ms); // TON
// fb_5_power(Enable := ton_en_5.Q, Axis := drive5); // MC_Power
// b_5_enable_on := fb_5_power.Status;

// NETWORK 26 (disabled)
//   b_enable_FI_6: the enable of drive 6
//   axisdata[6].Axis_InAb: A-0-0021.14 -RD- Axis is ready for power to the engine (Ab)
//   axisdata[6].Axis_Error: A-0-0021.09 -RD- Axis reports error
//   drive6: Real axis "Drive6" with axis number 6
// ton_en_6(IN := b_enable_FI_6 AND axisdata[6].Axis_InAb AND NOT axisdata[6].Axis_Error, PT := t#500ms); // TON
// fb_6_power(Enable := ton_en_6.Q, Axis := drive6); // MC_Power
// b_6_enable_on := fb_6_power.Status;

// NETWORK 27
//   axisdata[5].rActualPosition_i: A-0-0100 -RD- Actual position
//   v_FeedIndexer: Virtual axis "v_polarization" with axis number 9
// label: (*move FeedIndexer virtual axis to the position of driver 5*)
FB_move_master_FI(
    Execute := b_enable_FI_5,
    Position := axisdata[5].rActualPosition_i,
    Velocity := 10,
    Acceleration := 50,
    Deceleration := 50,
    Axis := v_FeedIndexer); // MC_MoveAbsolute
b_M_FI_done := FB_move_master_FI.Done;

// NETWORK 28 (disabled)
//   axisdata[5].Axis_Power: A-0-0021.15 -RD- Axis has power on (AH_AF)
//   axisdata[6].Axis_Power: A-0-0021.15 -RD- Axis has power on (AH_AF)
// label: (*change enable_on to AF*)
// b_home_FI2_done := NOT B_encoder_home_d5 AND b_encoder_ok_FI AND axisdata[5].Axis_Power AND axisdata[6].Axis_Power;

// NETWORK 29
//   axisdata[5].Axis_Power: A-0-0021.15 -RD- Axis has power on (AH_AF)
//   axisdata[6].Axis_Power: A-0-0021.15 -RD- Axis has power on (AH_AF)
// label: (*change enable_on to AF*)
b_home_FI2_done := axisdata[5].Axis_Power AND axisdata[6].Axis_Power AND b_enable_FI_5;

// NETWORK 30
//   v_FeedIndexer: Virtual axis "v_polarization" with axis number 9
//   drive5: Real axis "Drive5" with axis number 5
fb_gearinPos_FI(
    Execute := b_M_FI_done,
    RatioNumerator := 1,
    RatioDenominator := 1,
    MasterFineadjust := 0,
    SyncMode := 0,
    StartMode := 0,
    Master := v_FeedIndexer,
    Slave := drive5); // MB_GearInPos
b_gearin_5_done := fb_gearinPos_FI.InSync;

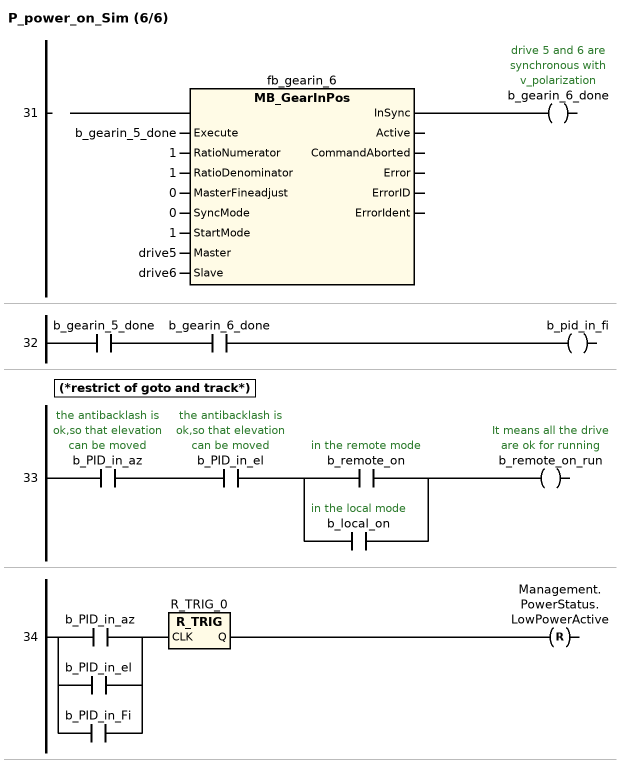
// NETWORK 31
//   drive5: Virtual axis "v_polarization" with axis number 9
//   drive6: Real axis "Drive6" with axis number 6
//   b_gearin_6_done: drive 5 and 6 are synchronous with v_polarization
fb_gearin_6(
    Execute := b_gearin_5_done,
    RatioNumerator := 1,
    RatioDenominator := 1,
    MasterFineadjust := 0,
    SyncMode := 0,
    StartMode := 1,
    Master := drive5,
    Slave := drive6); // MB_GearInPos
b_gearin_6_done := fb_gearin_6.InSync;

// NETWORK 32
b_pid_in_fi := b_gearin_5_done AND b_gearin_6_done;

// NETWORK 33
//   b_PID_in_az: the antibacklash is ok,so that elevation can be moved
//   b_PID_in_el: the antibacklash is ok,so that elevation can be moved
//   b_remote_on: in the remote mode
//   b_local_on: in the local mode
//   b_remote_on_run: It means all the drive are ok for running
// label: (*restrict of goto and track*)
b_remote_on_run := b_PID_in_az AND b_PID_in_el AND (b_remote_on OR b_local_on);

// NETWORK 34
R_TRIG_0(CLK := b_PID_in_az OR b_PID_in_el OR b_PID_in_Fi); // R_TRIG
Management.PowerStatus.LowPowerActive R= R_TRIG_0.Q;

END_PROGRAM

// IndraMotionMlc1/Application/POUs/Motion/P_power_off_TCP
(*the program is built for power off the 3 axis under the contol of remote or local.
the elevation axis is the similar with the azimuth*)
PROGRAM P_power_off_TCP
VAR
(*The firmware function block "MC_Stop" is used to bring the drive to the status STOP.*)
	fb_stop_v_az: MC_Stop;
	fb_stop_d1: MC_Stop;
	fb_stop_d2: MC_Stop;
	fb_stop_v_el: MC_Stop;
	fb_stop_d3: MC_Stop;
	fb_stop_d4: MC_Stop;
	fb_stop_v_FI: MC_Stop;
	fb_stop_d5: MC_Stop;
	fb_stop_d6: MC_Stop;
(*The firmware function block "MC_GearOut" is used to terminate an active synchronization function block.*)
	fb_gearout_d1: MC_GearOut;
	fb_gearout_d2: MC_GearOut;
	fb_gearout_d3: MC_GearOut;
	fb_gearout_d4: MC_GearOut;
	fb_gearout_d5: MC_GearOut;
	fb_gearout_d6: MC_GearOut;
(*The function block R_TRIG detects a rising edge*)
	rtrig_stop_az: R_TRIG;
	rtrig_stop_el: R_TRIG;
	rtrig_stop_FI: R_TRIG;
	rtrig_stop_d1: R_TRIG;
	rtrig_stop_d2: R_TRIG;
	rtrig_stop_d3: R_TRIG;
	rtrig_stop_d4: R_TRIG;
	rtrig_stop_d5: R_TRIG;
	rtrig_stop_d6: R_TRIG;
	rtrig_d1: R_TRIG;
	rtrig_d2: R_TRIG;
	rtrig_d3: R_TRIG;
	rtrig_d4: R_TRIG;
	rtrig_d5: R_TRIG;
	rtrig_d6: R_TRIG;
	rtrig_en_off: R_TRIG;
(*The function block F_TRIG a falling edge*)
	ftrig_reset_az: F_TRIG;
	ftrig_reset_el: F_TRIG;
	ftrig_reset_FI: F_TRIG;
(*The function block Timer On Delay implements a turn-on delay..*)
	fb_ton_powoff_az: TON;
	fb_ton_powoff_el: TON;
	fb_ton_powoff_FI: TON;
	fb_ton_en_off: TON;
	fb_ton_error: TON;
	FB_clear_all_error: MB_WriteParameter;
	fb_f_enable_off: F_TRIG;
	fb_R_enable_off: R_TRIG;
	fb_ton_enable_off: TON;
	b_enable_start: BOOL;
	fb_blink_reset: BLINK;
	b_clear_error: BOOL;
	fb_r_clear_error: R_TRIG;
	FB_clear_error_1: MB_WriteParameter;
	rtrig_clr_deactivate: R_TRIG;
	rtrig_el_deactivate_clear: R_TRIG;
	rtrig_deactivate_clear_el: R_TRIG;
	rtrig_clr_deactivate_az: R_TRIG;
	rtrig_clr_deactivate_fi: R_TRIG;
	b_execute_goto_Az: INT;
	b_start_goto_Az: BOOL;
END_VAR

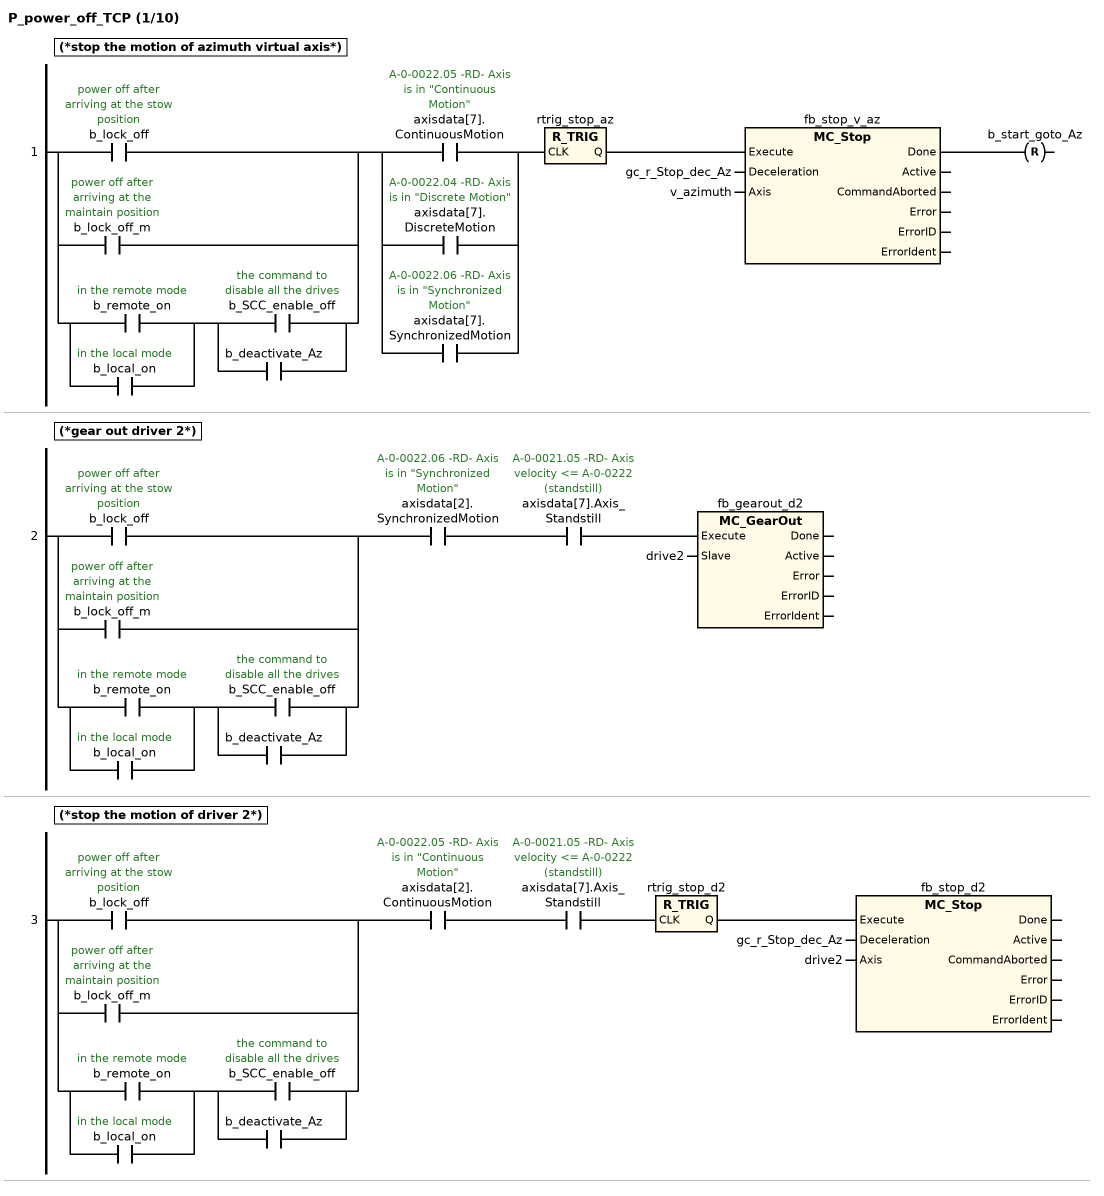
// NETWORK 1
//   fb_stop_v_az: The firmware function block "MC_Stop" is used to bring the drive to the status STOP.
//   rtrig_stop_az: The function block R_TRIG detects a rising edge
//   b_lock_off: power off after arriving at the stow position
//   b_lock_off_m: power off after arriving at the maintain position
//   b_remote_on: in the remote mode
//   b_local_on: in the local mode
//   b_SCC_enable_off: the command to disable all the drives
//   axisdata[7].ContinuousMotion: A-0-0022.05 -RD- Axis is in "Continuous Motion"
//   axisdata[7].DiscreteMotion: A-0-0022.04 -RD- Axis is in "Discrete Motion"
//   axisdata[7].SynchronizedMotion: A-0-0022.06 -RD- Axis is in "Synchronized Motion"
//   v_azimuth: Virtual axis "v_azimuth" with axis number 7
// label: (*stop the motion of azimuth virtual axis*)
rtrig_stop_az(CLK := (b_lock_off OR b_lock_off_m OR (b_remote_on OR b_local_on) AND (b_SCC_enable_off OR b_deactivate_Az)) AND (axisdata[7].ContinuousMotion OR axisdata[7].DiscreteMotion OR axisdata[7].SynchronizedMotion)); // R_TRIG
fb_stop_v_az(Execute := rtrig_stop_az.Q, Deceleration := gc_r_Stop_dec_Az, Axis := v_azimuth); // MC_Stop
b_start_goto_Az R= fb_stop_v_az.Done;

// NETWORK 2
//   b_lock_off: power off after arriving at the stow position
//   b_lock_off_m: power off after arriving at the maintain position
//   b_remote_on: in the remote mode
//   b_local_on: in the local mode
//   b_SCC_enable_off: the command to disable all the drives
//   axisdata[2].SynchronizedMotion: A-0-0022.06 -RD- Axis is in "Synchronized Motion"
//   axisdata[7].Axis_Standstill: A-0-0021.05 -RD- Axis velocity <= A-0-0222 (standstill)
//   drive2: Real axis "Drive2" with axis number 2
// label: (*gear out driver 2*)
fb_gearout_d2(Execute := (b_lock_off OR b_lock_off_m OR (b_remote_on OR b_local_on) AND (b_SCC_enable_off OR b_deactivate_Az)) AND axisdata[2].SynchronizedMotion AND axisdata[7].Axis_Standstill, Slave := drive2); // MC_GearOut

// NETWORK 3
//   b_lock_off: power off after arriving at the stow position
//   b_lock_off_m: power off after arriving at the maintain position
//   b_remote_on: in the remote mode
//   b_local_on: in the local mode
//   b_SCC_enable_off: the command to disable all the drives
//   axisdata[2].ContinuousMotion: A-0-0022.05 -RD- Axis is in "Continuous Motion"
//   axisdata[7].Axis_Standstill: A-0-0021.05 -RD- Axis velocity <= A-0-0222 (standstill)
//   drive2: Real axis "Drive2" with axis number 2
// label: (*stop the motion of driver 2*)
rtrig_stop_d2(CLK := (b_lock_off OR b_lock_off_m OR (b_remote_on OR b_local_on) AND (b_SCC_enable_off OR b_deactivate_Az)) AND axisdata[2].ContinuousMotion AND axisdata[7].Axis_Standstill); // R_TRIG
fb_stop_d2(Execute := rtrig_stop_d2.Q, Deceleration := gc_r_Stop_dec_Az, Axis := drive2); // MC_Stop

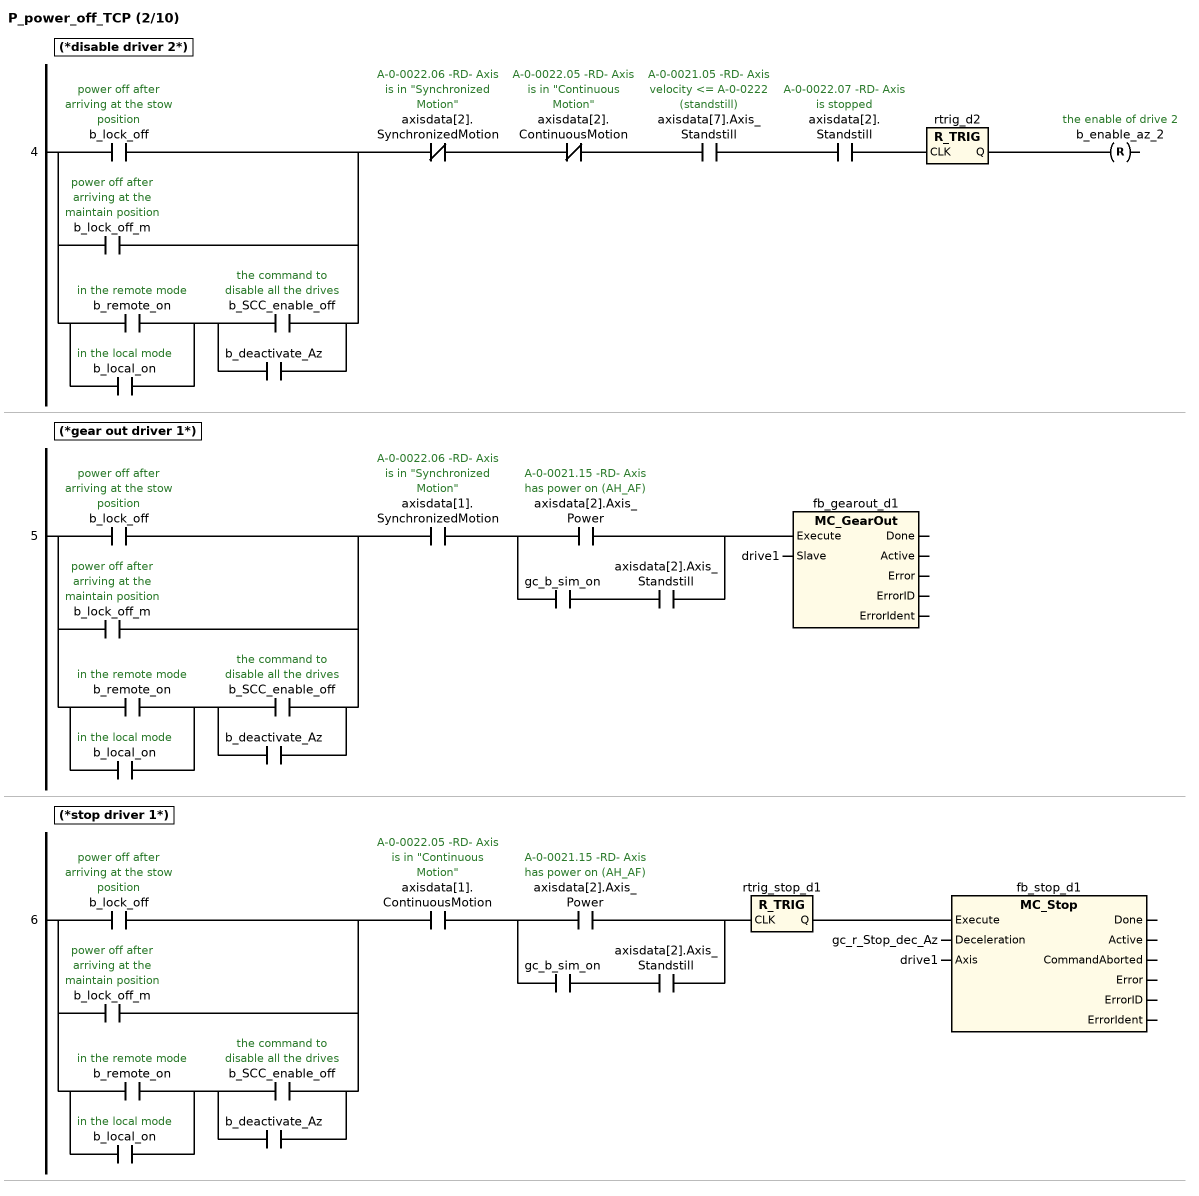
// NETWORK 4
//   b_lock_off: power off after arriving at the stow position
//   b_lock_off_m: power off after arriving at the maintain position
//   b_remote_on: in the remote mode
//   b_local_on: in the local mode
//   b_SCC_enable_off: the command to disable all the drives
//   axisdata[2].SynchronizedMotion: A-0-0022.06 -RD- Axis is in "Synchronized Motion"
//   axisdata[2].ContinuousMotion: A-0-0022.05 -RD- Axis is in "Continuous Motion"
//   axisdata[7].Axis_Standstill: A-0-0021.05 -RD- Axis velocity <= A-0-0222 (standstill)
//   axisdata[2].Standstill: A-0-0022.07 -RD- Axis is stopped
//   b_enable_az_2: the enable of drive 2
// label: (*disable driver 2*)
rtrig_d2(CLK := (b_lock_off OR b_lock_off_m OR (b_remote_on OR b_local_on) AND (b_SCC_enable_off OR b_deactivate_Az)) AND NOT axisdata[2].SynchronizedMotion AND NOT axisdata[2].ContinuousMotion AND axisdata[7].Axis_Standstill AND axisdata[2].Standstill); // R_TRIG
b_enable_az_2 R= rtrig_d2.Q;

// NETWORK 5
//   fb_gearout_d1: The firmware function block "MC_GearOut" is used to terminate an active synchronization function block.
//   b_lock_off: power off after arriving at the stow position
//   b_lock_off_m: power off after arriving at the maintain position
//   b_remote_on: in the remote mode
//   b_local_on: in the local mode
//   b_SCC_enable_off: the command to disable all the drives
//   axisdata[1].SynchronizedMotion: A-0-0022.06 -RD- Axis is in "Synchronized Motion"
//   axisdata[2].Axis_Power: A-0-0021.15 -RD- Axis has power on (AH_AF)
//   drive1: Real axis "Drive1" with axis number 1
// label: (*gear out driver 1*)
fb_gearout_d1(Execute := (b_lock_off OR b_lock_off_m OR (b_remote_on OR b_local_on) AND (b_SCC_enable_off OR b_deactivate_Az)) AND axisdata[1].SynchronizedMotion AND (axisdata[2].Axis_Power OR gc_b_sim_on AND axisdata[2].Axis_Standstill), Slave := drive1); // MC_GearOut

// NETWORK 6
//   b_lock_off: power off after arriving at the stow position
//   b_lock_off_m: power off after arriving at the maintain position
//   b_remote_on: in the remote mode
//   b_local_on: in the local mode
//   b_SCC_enable_off: the command to disable all the drives
//   axisdata[1].ContinuousMotion: A-0-0022.05 -RD- Axis is in "Continuous Motion"
//   axisdata[2].Axis_Power: A-0-0021.15 -RD- Axis has power on (AH_AF)
//   drive1: Real axis "Drive1" with axis number 1
// label: (*stop driver 1*)
rtrig_stop_d1(CLK := (b_lock_off OR b_lock_off_m OR (b_remote_on OR b_local_on) AND (b_SCC_enable_off OR b_deactivate_Az)) AND axisdata[1].ContinuousMotion AND (axisdata[2].Axis_Power OR gc_b_sim_on AND axisdata[2].Axis_Standstill)); // R_TRIG
fb_stop_d1(Execute := rtrig_stop_d1.Q, Deceleration := gc_r_Stop_dec_Az, Axis := drive1); // MC_Stop

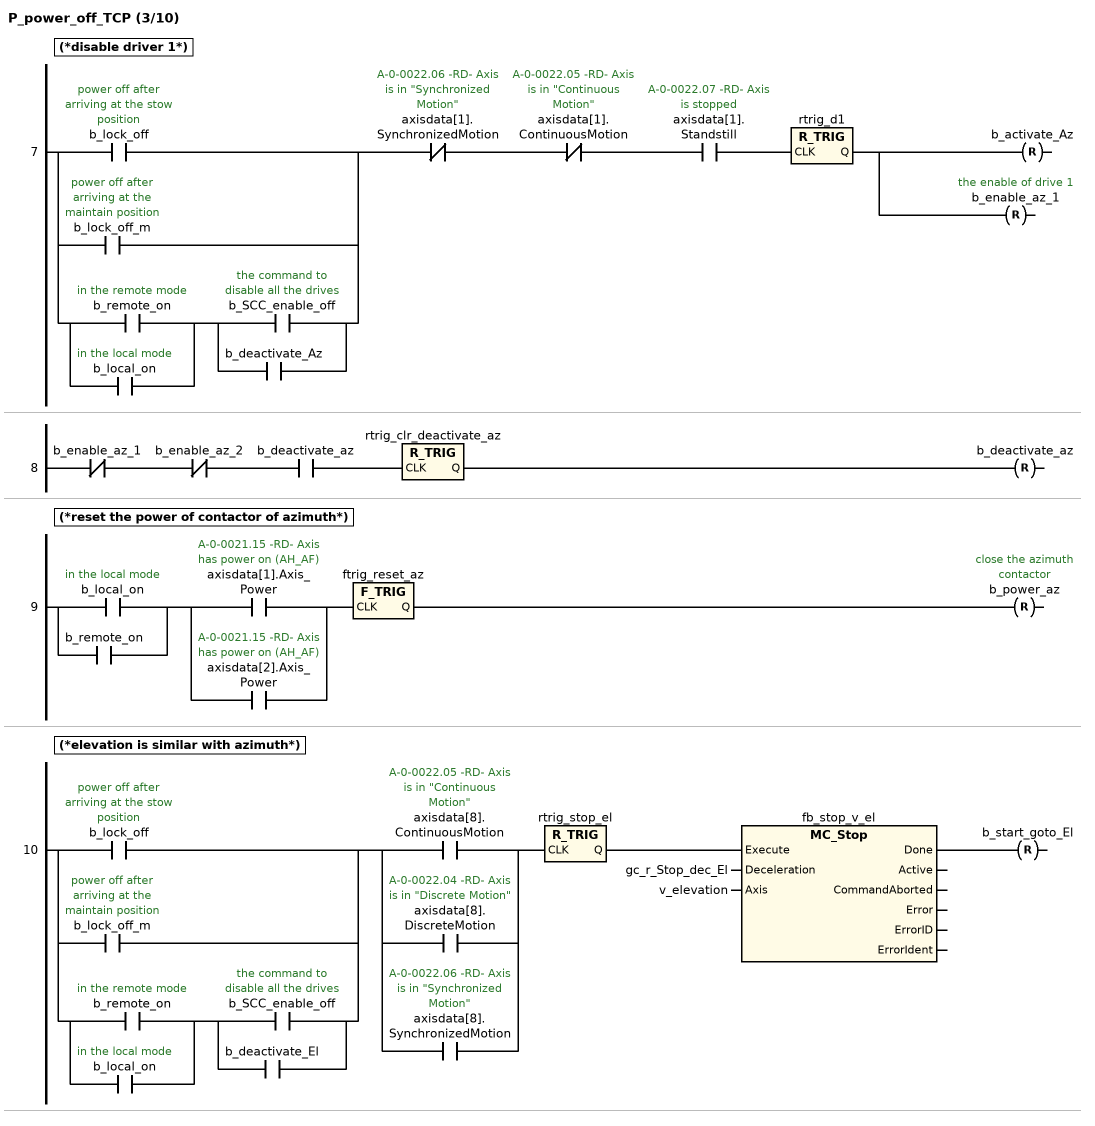
// NETWORK 7
//   b_lock_off: power off after arriving at the stow position
//   b_lock_off_m: power off after arriving at the maintain position
//   b_remote_on: in the remote mode
//   b_local_on: in the local mode
//   b_SCC_enable_off: the command to disable all the drives
//   axisdata[1].SynchronizedMotion: A-0-0022.06 -RD- Axis is in "Synchronized Motion"
//   axisdata[1].ContinuousMotion: A-0-0022.05 -RD- Axis is in "Continuous Motion"
//   axisdata[1].Standstill: A-0-0022.07 -RD- Axis is stopped
//   b_enable_az_1: the enable of drive 1
// label: (*disable driver 1*)
rtrig_d1(CLK := (b_lock_off OR b_lock_off_m OR (b_remote_on OR b_local_on) AND (b_SCC_enable_off OR b_deactivate_Az)) AND NOT axisdata[1].SynchronizedMotion AND NOT axisdata[1].ContinuousMotion AND axisdata[1].Standstill); // R_TRIG
b_activate_Az R= rtrig_d1.Q;
b_enable_az_1 R= rtrig_d1.Q;

// NETWORK 8
rtrig_clr_deactivate_az(CLK := NOT b_enable_az_1 AND NOT b_enable_az_2 AND b_deactivate_az); // R_TRIG
b_deactivate_az R= rtrig_clr_deactivate_az.Q;

// NETWORK 9
//   ftrig_reset_az: The function block F_TRIG a falling edge
//   b_local_on: in the local mode
//   axisdata[1].Axis_Power: A-0-0021.15 -RD- Axis has power on (AH_AF)
//   axisdata[2].Axis_Power: A-0-0021.15 -RD- Axis has power on (AH_AF)
//   b_power_az: close the azimuth contactor
// label: (*reset the power of contactor of azimuth*)
ftrig_reset_az(CLK := (b_local_on OR b_remote_on) AND (axisdata[1].Axis_Power OR axisdata[2].Axis_Power)); // F_TRIG
b_power_az R= ftrig_reset_az.Q;

// NETWORK 10
//   b_lock_off: power off after arriving at the stow position
//   b_lock_off_m: power off after arriving at the maintain position
//   b_remote_on: in the remote mode
//   b_local_on: in the local mode
//   b_SCC_enable_off: the command to disable all the drives
//   axisdata[8].ContinuousMotion: A-0-0022.05 -RD- Axis is in "Continuous Motion"
//   axisdata[8].DiscreteMotion: A-0-0022.04 -RD- Axis is in "Discrete Motion"
//   axisdata[8].SynchronizedMotion: A-0-0022.06 -RD- Axis is in "Synchronized Motion"
//   v_elevation: Virtual axis "v_elevation" with axis number 8
// label: (*elevation is similar with azimuth*)
rtrig_stop_el(CLK := (b_lock_off OR b_lock_off_m OR (b_remote_on OR b_local_on) AND (b_SCC_enable_off OR b_deactivate_El)) AND (axisdata[8].ContinuousMotion OR axisdata[8].DiscreteMotion OR axisdata[8].SynchronizedMotion)); // R_TRIG
fb_stop_v_el(Execute := rtrig_stop_el.Q, Deceleration := gc_r_Stop_dec_El, Axis := v_elevation); // MC_Stop
b_start_goto_El R= fb_stop_v_el.Done;

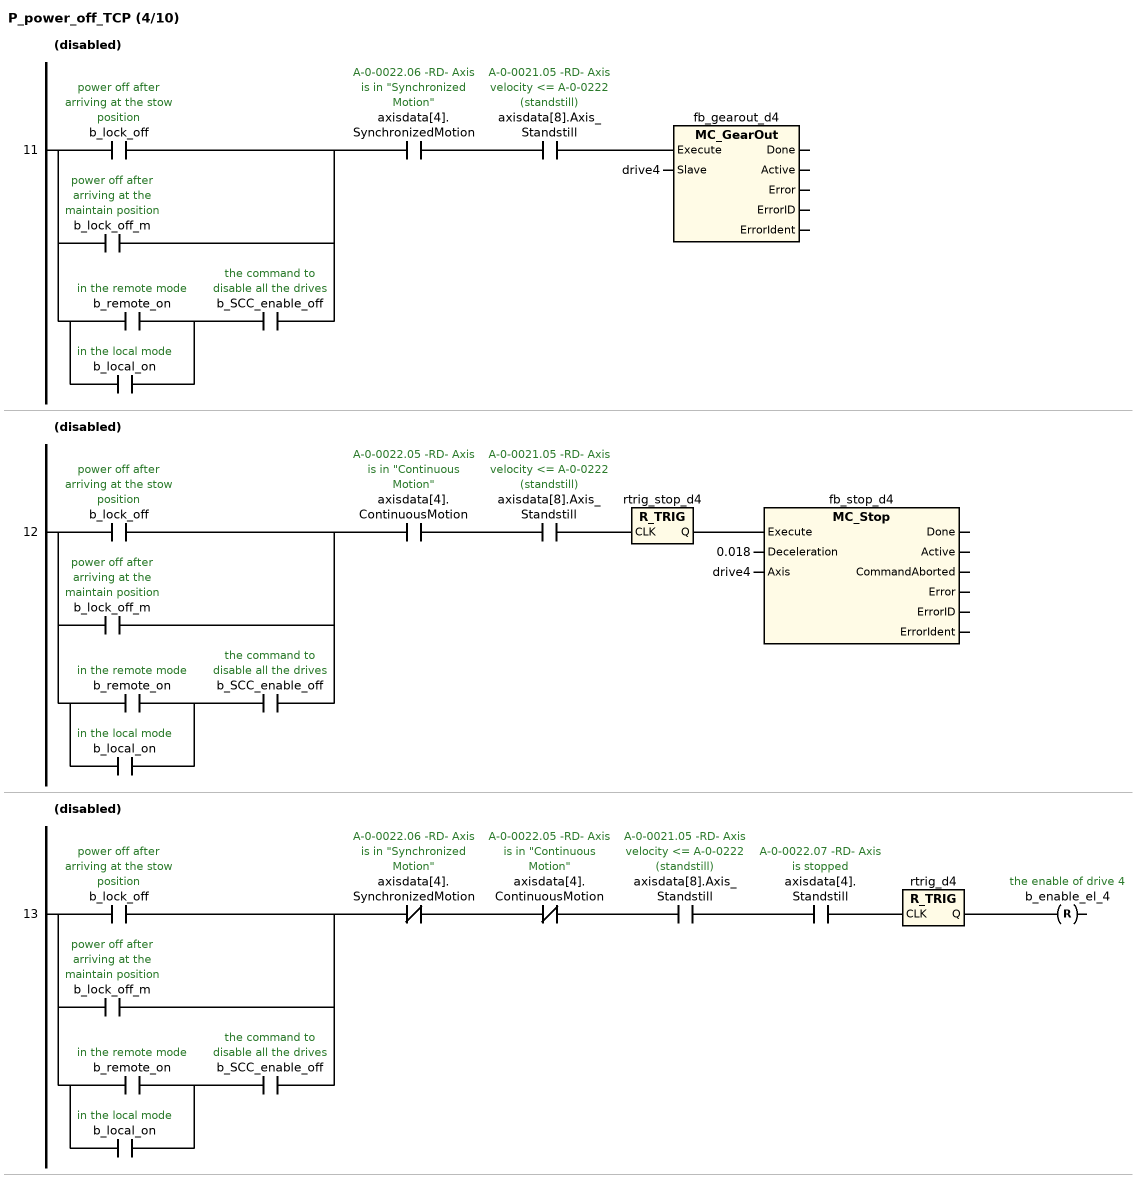
// NETWORK 11 (disabled)
//   b_lock_off: power off after arriving at the stow position
//   b_lock_off_m: power off after arriving at the maintain position
//   b_remote_on: in the remote mode
//   b_local_on: in the local mode
//   b_SCC_enable_off: the command to disable all the drives
//   axisdata[4].SynchronizedMotion: A-0-0022.06 -RD- Axis is in "Synchronized Motion"
//   axisdata[8].Axis_Standstill: A-0-0021.05 -RD- Axis velocity <= A-0-0222 (standstill)
//   drive4: Real axis "Drive4" with axis number 4
// fb_gearout_d4(Execute := (b_lock_off OR b_lock_off_m OR (b_remote_on OR b_local_on) AND b_SCC_enable_off) AND axisdata[4].SynchronizedMotion AND axisdata[8].Axis_Standstill, Slave := drive4); // MC_GearOut

// NETWORK 12 (disabled)
//   b_lock_off: power off after arriving at the stow position
//   b_lock_off_m: power off after arriving at the maintain position
//   b_remote_on: in the remote mode
//   b_local_on: in the local mode
//   b_SCC_enable_off: the command to disable all the drives
//   axisdata[4].ContinuousMotion: A-0-0022.05 -RD- Axis is in "Continuous Motion"
//   axisdata[8].Axis_Standstill: A-0-0021.05 -RD- Axis velocity <= A-0-0222 (standstill)
//   drive4: Real axis "Drive4" with axis number 4
// rtrig_stop_d4(CLK := (b_lock_off OR b_lock_off_m OR (b_remote_on OR b_local_on) AND b_SCC_enable_off) AND axisdata[4].ContinuousMotion AND axisdata[8].Axis_Standstill); // R_TRIG
// fb_stop_d4(Execute := rtrig_stop_d4.Q, Deceleration := 0.018, Axis := drive4); // MC_Stop

// NETWORK 13 (disabled)
//   b_lock_off: power off after arriving at the stow position
//   b_lock_off_m: power off after arriving at the maintain position
//   b_remote_on: in the remote mode
//   b_local_on: in the local mode
//   b_SCC_enable_off: the command to disable all the drives
//   axisdata[4].SynchronizedMotion: A-0-0022.06 -RD- Axis is in "Synchronized Motion"
//   axisdata[4].ContinuousMotion: A-0-0022.05 -RD- Axis is in "Continuous Motion"
//   axisdata[8].Axis_Standstill: A-0-0021.05 -RD- Axis velocity <= A-0-0222 (standstill)
//   axisdata[4].Standstill: A-0-0022.07 -RD- Axis is stopped
//   b_enable_el_4: the enable of drive 4
// rtrig_d4(CLK := (b_lock_off OR b_lock_off_m OR (b_remote_on OR b_local_on) AND b_SCC_enable_off) AND NOT axisdata[4].SynchronizedMotion AND NOT axisdata[4].ContinuousMotion AND axisdata[8].Axis_Standstill AND axisdata[4].Standstill); // R_TRIG
// b_enable_el_4 R= rtrig_d4.Q;

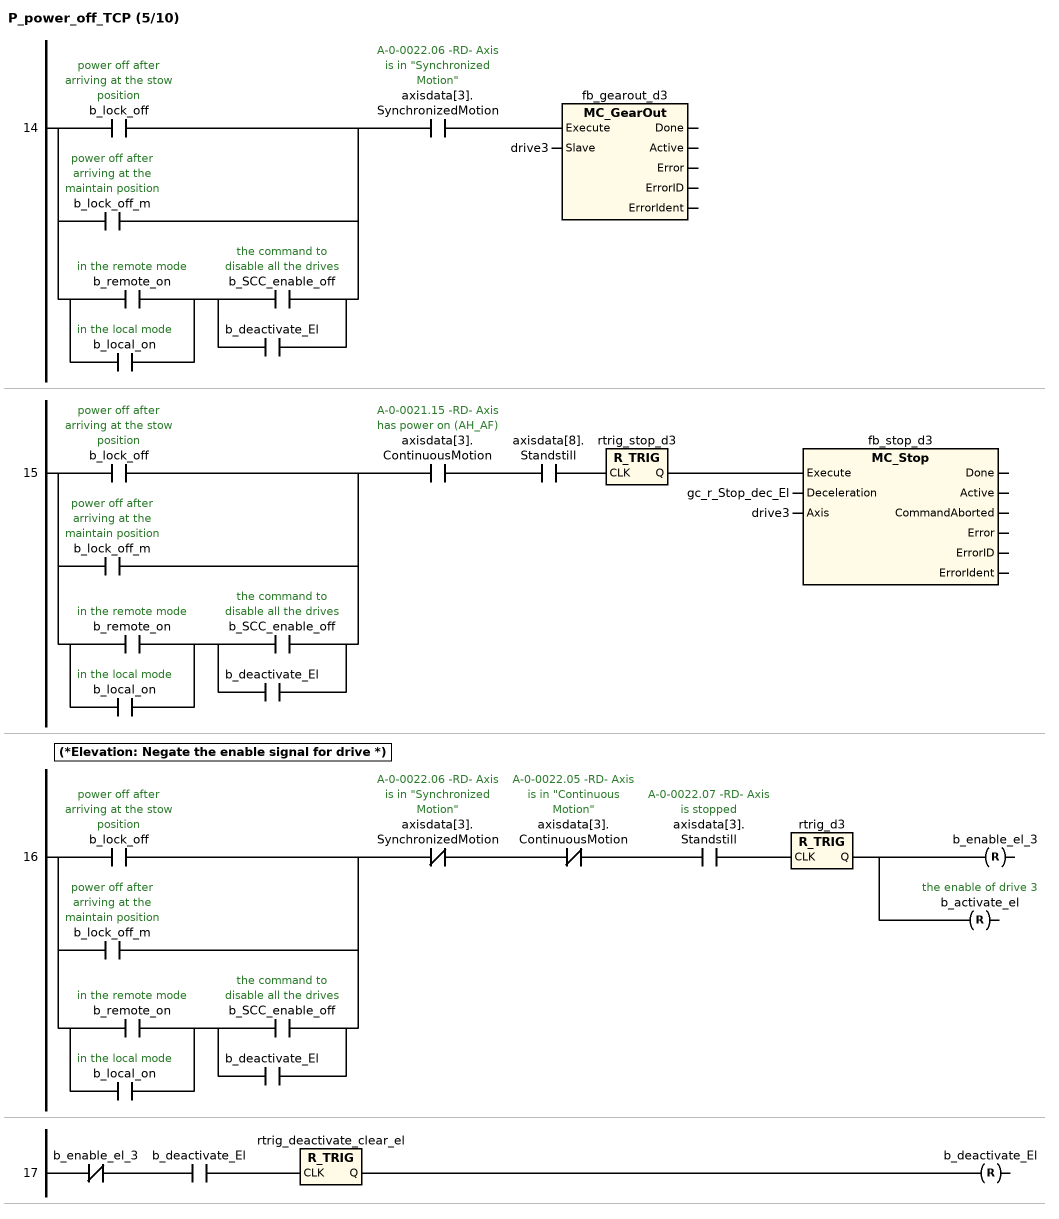
// NETWORK 14
//   b_lock_off: power off after arriving at the stow position
//   b_lock_off_m: power off after arriving at the maintain position
//   b_remote_on: in the remote mode
//   b_local_on: in the local mode
//   b_SCC_enable_off: the command to disable all the drives
//   axisdata[3].SynchronizedMotion: A-0-0022.06 -RD- Axis is in "Synchronized Motion"
//   drive3: Real axis "Drive3" with axis number 3
fb_gearout_d3(Execute := (b_lock_off OR b_lock_off_m OR (b_remote_on OR b_local_on) AND (b_SCC_enable_off OR b_deactivate_El)) AND axisdata[3].SynchronizedMotion, Slave := drive3); // MC_GearOut

// NETWORK 15
//   b_lock_off: power off after arriving at the stow position
//   b_lock_off_m: power off after arriving at the maintain position
//   b_remote_on: in the remote mode
//   b_local_on: in the local mode
//   b_SCC_enable_off: the command to disable all the drives
//   axisdata[3].ContinuousMotion: A-0-0021.15 -RD- Axis has power on (AH_AF)
//   drive3: Real axis "Drive3" with axis number 3
rtrig_stop_d3(CLK := (b_lock_off OR b_lock_off_m OR (b_remote_on OR b_local_on) AND (b_SCC_enable_off OR b_deactivate_El)) AND axisdata[3].ContinuousMotion AND axisdata[8].Standstill); // R_TRIG
fb_stop_d3(Execute := rtrig_stop_d3.Q, Deceleration := gc_r_Stop_dec_El, Axis := drive3); // MC_Stop

// NETWORK 16
//   b_lock_off: power off after arriving at the stow position
//   b_lock_off_m: power off after arriving at the maintain position
//   b_remote_on: in the remote mode
//   b_local_on: in the local mode
//   b_SCC_enable_off: the command to disable all the drives
//   axisdata[3].SynchronizedMotion: A-0-0022.06 -RD- Axis is in "Synchronized Motion"
//   axisdata[3].ContinuousMotion: A-0-0022.05 -RD- Axis is in "Continuous Motion"
//   axisdata[3].Standstill: A-0-0022.07 -RD- Axis is stopped
//   b_activate_el: the enable of drive 3
// label: (*Elevation: Negate the enable signal for drive *)
rtrig_d3(CLK := (b_lock_off OR b_lock_off_m OR (b_remote_on OR b_local_on) AND (b_SCC_enable_off OR b_deactivate_El)) AND NOT axisdata[3].SynchronizedMotion AND NOT axisdata[3].ContinuousMotion AND axisdata[3].Standstill); // R_TRIG
b_enable_el_3 R= rtrig_d3.Q;
b_activate_el R= rtrig_d3.Q;

// NETWORK 17
rtrig_deactivate_clear_el(CLK := NOT b_enable_el_3 AND b_deactivate_El); // R_TRIG
b_deactivate_El R= rtrig_deactivate_clear_el.Q;

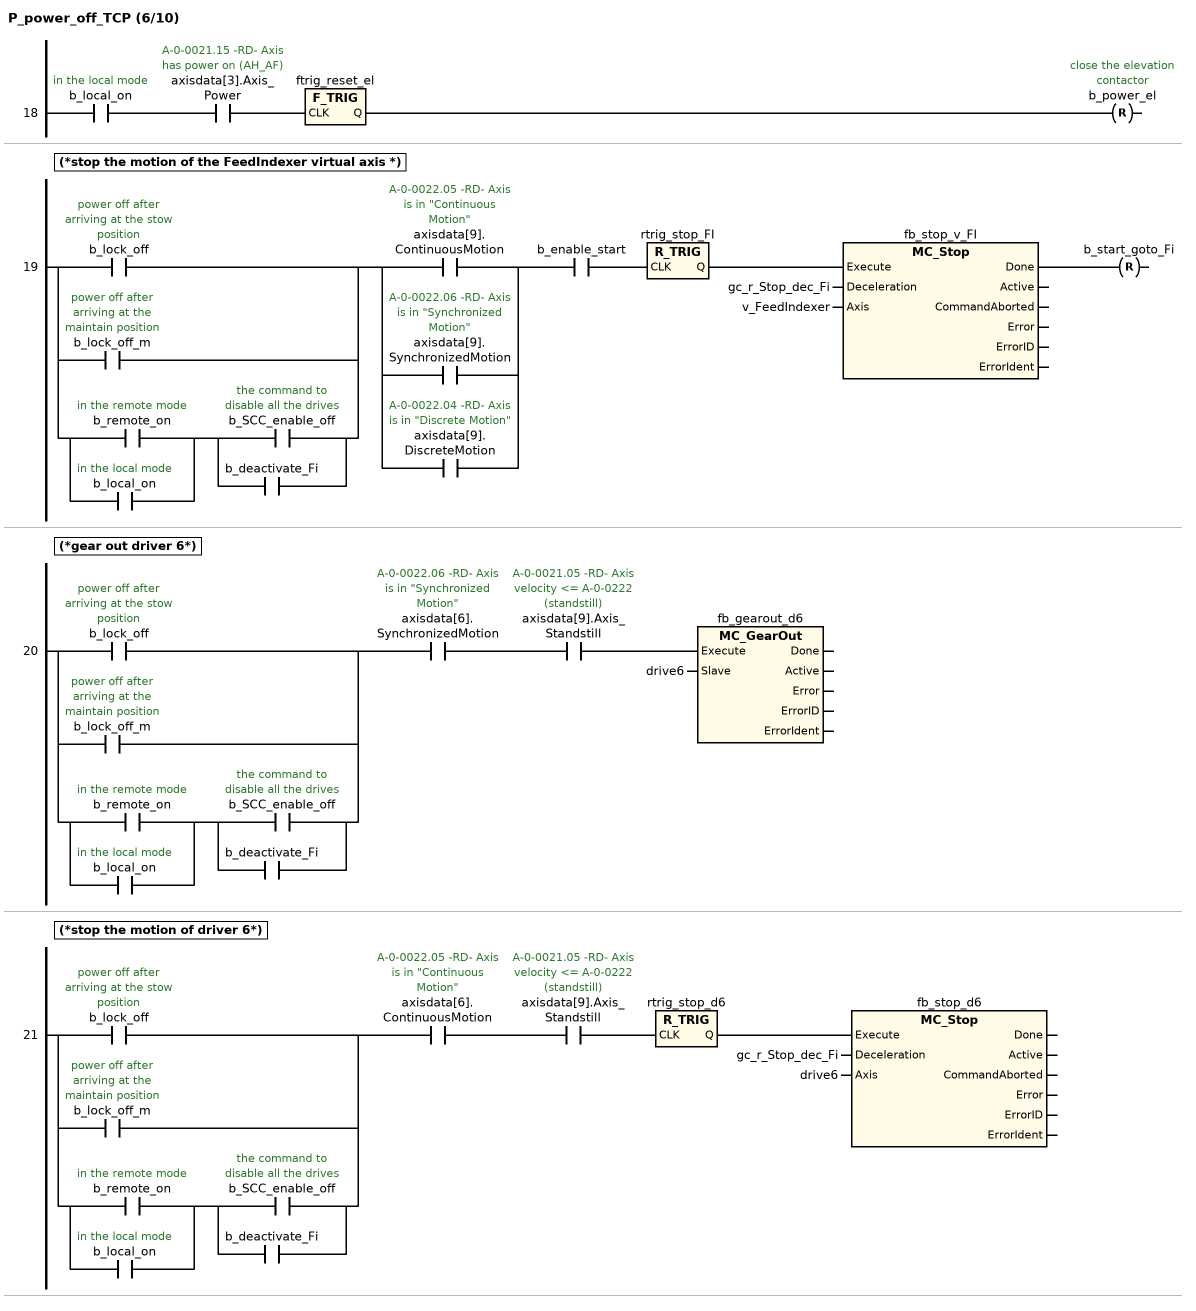
// NETWORK 18
//   b_local_on: in the local mode
//   axisdata[3].Axis_Power: A-0-0021.15 -RD- Axis has power on (AH_AF)
//   b_power_el: close the elevation contactor
ftrig_reset_el(CLK := b_local_on AND axisdata[3].Axis_Power); // F_TRIG
b_power_el R= ftrig_reset_el.Q;

// NETWORK 19
//   b_lock_off: power off after arriving at the stow position
//   b_lock_off_m: power off after arriving at the maintain position
//   b_remote_on: in the remote mode
//   b_local_on: in the local mode
//   b_SCC_enable_off: the command to disable all the drives
//   axisdata[9].ContinuousMotion: A-0-0022.05 -RD- Axis is in "Continuous Motion"
//   axisdata[9].SynchronizedMotion: A-0-0022.06 -RD- Axis is in "Synchronized Motion"
//   axisdata[9].DiscreteMotion: A-0-0022.04 -RD- Axis is in "Discrete Motion"
//   v_FeedIndexer: Virtual axis "v_polarization" with axis number 9
// label: (*stop the motion of the FeedIndexer virtual axis *)
rtrig_stop_FI(CLK := (b_lock_off OR b_lock_off_m OR (b_remote_on OR b_local_on) AND (b_SCC_enable_off OR b_deactivate_Fi)) AND (axisdata[9].ContinuousMotion OR axisdata[9].SynchronizedMotion OR axisdata[9].DiscreteMotion) AND b_enable_start); // R_TRIG
fb_stop_v_FI(Execute := rtrig_stop_FI.Q, Deceleration := gc_r_Stop_dec_Fi, Axis := v_FeedIndexer); // MC_Stop
b_start_goto_Fi R= fb_stop_v_FI.Done;

// NETWORK 20
//   b_lock_off: power off after arriving at the stow position
//   b_lock_off_m: power off after arriving at the maintain position
//   b_remote_on: in the remote mode
//   b_local_on: in the local mode
//   b_SCC_enable_off: the command to disable all the drives
//   axisdata[6].SynchronizedMotion: A-0-0022.06 -RD- Axis is in "Synchronized Motion"
//   axisdata[9].Axis_Standstill: A-0-0021.05 -RD- Axis velocity <= A-0-0222 (standstill)
//   drive6: Real axis "Drive6" with axis number 6
// label: (*gear out driver 6*)
fb_gearout_d6(Execute := (b_lock_off OR b_lock_off_m OR (b_remote_on OR b_local_on) AND (b_SCC_enable_off OR b_deactivate_Fi)) AND axisdata[6].SynchronizedMotion AND axisdata[9].Axis_Standstill, Slave := drive6); // MC_GearOut

// NETWORK 21
//   b_lock_off: power off after arriving at the stow position
//   b_lock_off_m: power off after arriving at the maintain position
//   b_remote_on: in the remote mode
//   b_local_on: in the local mode
//   b_SCC_enable_off: the command to disable all the drives
//   axisdata[6].ContinuousMotion: A-0-0022.05 -RD- Axis is in "Continuous Motion"
//   axisdata[9].Axis_Standstill: A-0-0021.05 -RD- Axis velocity <= A-0-0222 (standstill)
//   drive6: Real axis "Drive6" with axis number 6
// label: (*stop the motion of driver 6*)
rtrig_stop_d6(CLK := (b_lock_off OR b_lock_off_m OR (b_remote_on OR b_local_on) AND (b_SCC_enable_off OR b_deactivate_Fi)) AND axisdata[6].ContinuousMotion AND axisdata[9].Axis_Standstill); // R_TRIG
fb_stop_d6(Execute := rtrig_stop_d6.Q, Deceleration := gc_r_Stop_dec_Fi, Axis := drive6); // MC_Stop

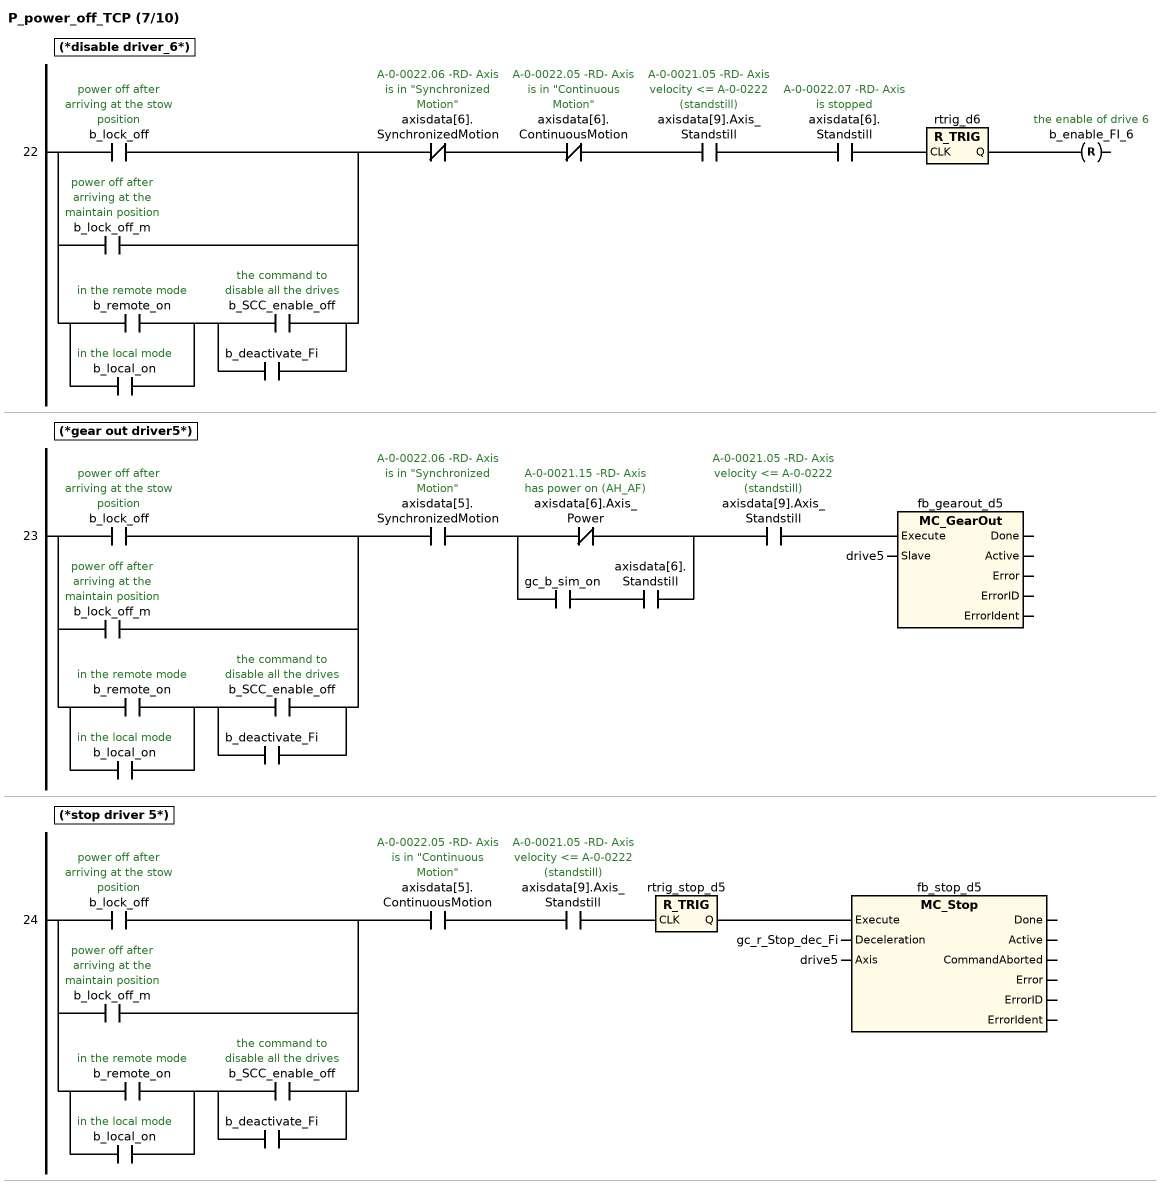
// NETWORK 22
//   b_lock_off: power off after arriving at the stow position
//   b_lock_off_m: power off after arriving at the maintain position
//   b_remote_on: in the remote mode
//   b_local_on: in the local mode
//   b_SCC_enable_off: the command to disable all the drives
//   axisdata[6].SynchronizedMotion: A-0-0022.06 -RD- Axis is in "Synchronized Motion"
//   axisdata[6].ContinuousMotion: A-0-0022.05 -RD- Axis is in "Continuous Motion"
//   axisdata[9].Axis_Standstill: A-0-0021.05 -RD- Axis velocity <= A-0-0222 (standstill)
//   axisdata[6].Standstill: A-0-0022.07 -RD- Axis is stopped
//   b_enable_FI_6: the enable of drive 6
// label: (*disable driver_6*)
rtrig_d6(CLK := (b_lock_off OR b_lock_off_m OR (b_remote_on OR b_local_on) AND (b_SCC_enable_off OR b_deactivate_Fi)) AND NOT axisdata[6].SynchronizedMotion AND NOT axisdata[6].ContinuousMotion AND axisdata[9].Axis_Standstill AND axisdata[6].Standstill); // R_TRIG
b_enable_FI_6 R= rtrig_d6.Q;

// NETWORK 23
//   b_lock_off: power off after arriving at the stow position
//   b_lock_off_m: power off after arriving at the maintain position
//   b_remote_on: in the remote mode
//   b_local_on: in the local mode
//   b_SCC_enable_off: the command to disable all the drives
//   axisdata[5].SynchronizedMotion: A-0-0022.06 -RD- Axis is in "Synchronized Motion"
//   axisdata[6].Axis_Power: A-0-0021.15 -RD- Axis has power on (AH_AF)
//   axisdata[9].Axis_Standstill: A-0-0021.05 -RD- Axis velocity <= A-0-0222 (standstill)
//   drive5: Real axis "Drive5" with axis number 5
// label: (*gear out driver5*)
fb_gearout_d5(Execute := (b_lock_off OR b_lock_off_m OR (b_remote_on OR b_local_on) AND (b_SCC_enable_off OR b_deactivate_Fi)) AND axisdata[5].SynchronizedMotion AND (NOT axisdata[6].Axis_Power OR gc_b_sim_on AND axisdata[6].Standstill) AND axisdata[9].Axis_Standstill, Slave := drive5); // MC_GearOut

// NETWORK 24
//   b_lock_off: power off after arriving at the stow position
//   b_lock_off_m: power off after arriving at the maintain position
//   b_remote_on: in the remote mode
//   b_local_on: in the local mode
//   b_SCC_enable_off: the command to disable all the drives
//   axisdata[5].ContinuousMotion: A-0-0022.05 -RD- Axis is in "Continuous Motion"
//   axisdata[9].Axis_Standstill: A-0-0021.05 -RD- Axis velocity <= A-0-0222 (standstill)
//   drive5: Real axis "Drive5" with axis number 5
// label: (*stop driver 5*)
rtrig_stop_d5(CLK := (b_lock_off OR b_lock_off_m OR (b_remote_on OR b_local_on) AND (b_SCC_enable_off OR b_deactivate_Fi)) AND axisdata[5].ContinuousMotion AND axisdata[9].Axis_Standstill); // R_TRIG
fb_stop_d5(Execute := rtrig_stop_d5.Q, Deceleration := gc_r_Stop_dec_Fi, Axis := drive5); // MC_Stop

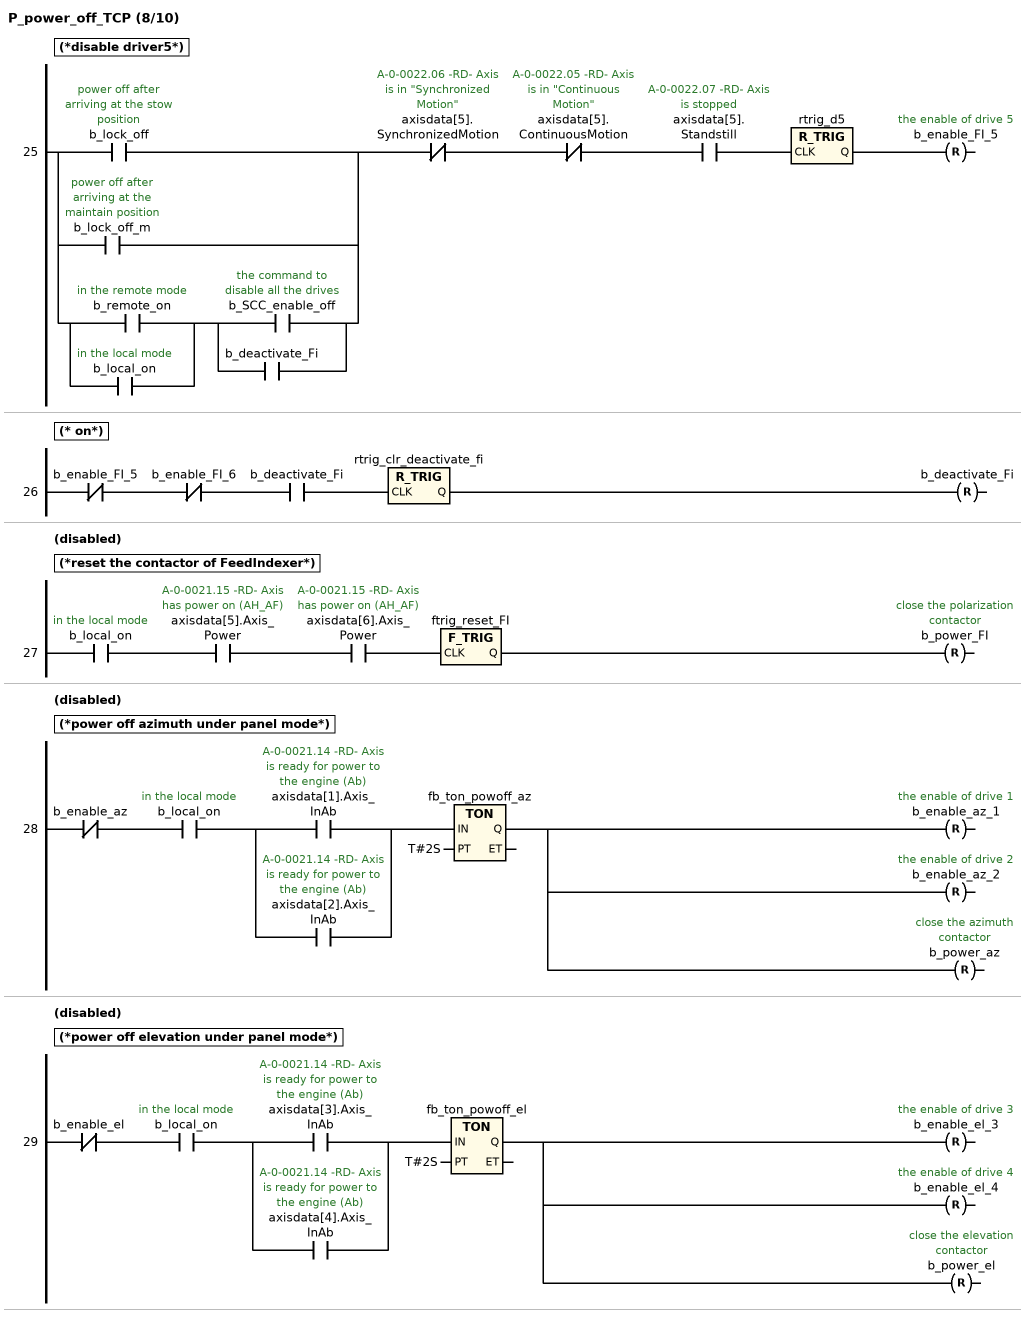
// NETWORK 25
//   b_lock_off: power off after arriving at the stow position
//   b_lock_off_m: power off after arriving at the maintain position
//   b_remote_on: in the remote mode
//   b_local_on: in the local mode
//   b_SCC_enable_off: the command to disable all the drives
//   axisdata[5].SynchronizedMotion: A-0-0022.06 -RD- Axis is in "Synchronized Motion"
//   axisdata[5].ContinuousMotion: A-0-0022.05 -RD- Axis is in "Continuous Motion"
//   axisdata[5].Standstill: A-0-0022.07 -RD- Axis is stopped
//   b_enable_FI_5: the enable of drive 5
// label: (*disable driver5*)
rtrig_d5(CLK := (b_lock_off OR b_lock_off_m OR (b_remote_on OR b_local_on) AND (b_SCC_enable_off OR b_deactivate_Fi)) AND NOT axisdata[5].SynchronizedMotion AND NOT axisdata[5].ContinuousMotion AND axisdata[5].Standstill); // R_TRIG
b_enable_FI_5 R= rtrig_d5.Q;

// NETWORK 26
// label: (* on*)
rtrig_clr_deactivate_fi(CLK := NOT b_enable_FI_5 AND NOT b_enable_FI_6 AND b_deactivate_Fi); // R_TRIG
b_deactivate_Fi R= rtrig_clr_deactivate_fi.Q;

// NETWORK 27 (disabled)
//   b_local_on: in the local mode
//   axisdata[5].Axis_Power: A-0-0021.15 -RD- Axis has power on (AH_AF)
//   axisdata[6].Axis_Power: A-0-0021.15 -RD- Axis has power on (AH_AF)
//   b_power_FI: close the polarization contactor
// label: (*reset the contactor of FeedIndexer*)
// ftrig_reset_FI(CLK := b_local_on AND axisdata[5].Axis_Power AND axisdata[6].Axis_Power); // F_TRIG
// b_power_FI R= ftrig_reset_FI.Q;

// NETWORK 28 (disabled)
//   fb_ton_powoff_az: The function block Timer On Delay implements a turn-on delay..
//   b_local_on: in the local mode
//   axisdata[1].Axis_InAb: A-0-0021.14 -RD- Axis is ready for power to the engine (Ab)
//   axisdata[2].Axis_InAb: A-0-0021.14 -RD- Axis is ready for power to the engine (Ab)
//   b_enable_az_1: the enable of drive 1
//   b_enable_az_2: the enable of drive 2
//   b_power_az: close the azimuth contactor
// label: (*power off azimuth under panel mode*)
// fb_ton_powoff_az(IN := NOT b_enable_az AND b_local_on AND (axisdata[1].Axis_InAb OR axisdata[2].Axis_InAb), PT := T#2S); // TON
// b_enable_az_1 R= fb_ton_powoff_az.Q;
// b_enable_az_2 R= fb_ton_powoff_az.Q;
// b_power_az R= fb_ton_powoff_az.Q;

// NETWORK 29 (disabled)
//   b_local_on: in the local mode
//   axisdata[3].Axis_InAb: A-0-0021.14 -RD- Axis is ready for power to the engine (Ab)
//   axisdata[4].Axis_InAb: A-0-0021.14 -RD- Axis is ready for power to the engine (Ab)
//   b_enable_el_3: the enable of drive 3
//   b_enable_el_4: the enable of drive 4
//   b_power_el: close the elevation contactor
// label: (*power off elevation under panel mode*)
// fb_ton_powoff_el(IN := NOT b_enable_el AND b_local_on AND (axisdata[3].Axis_InAb OR axisdata[4].Axis_InAb), PT := T#2S); // TON
// b_enable_el_3 R= fb_ton_powoff_el.Q;
// b_enable_el_4 R= fb_ton_powoff_el.Q;
// b_power_el R= fb_ton_powoff_el.Q;

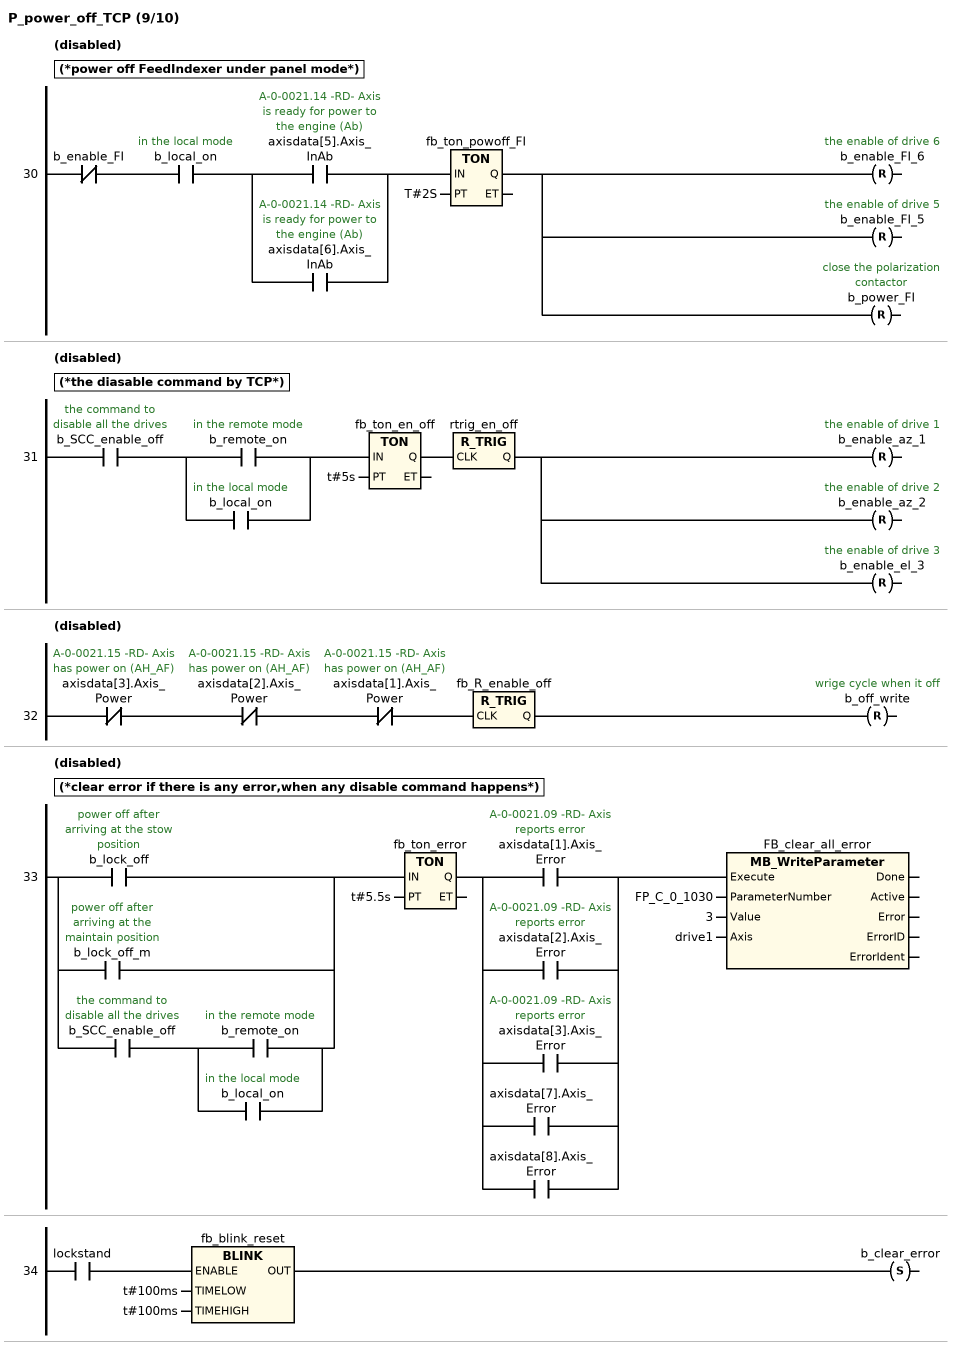
// NETWORK 30 (disabled)
//   b_local_on: in the local mode
//   axisdata[5].Axis_InAb: A-0-0021.14 -RD- Axis is ready for power to the engine (Ab)
//   axisdata[6].Axis_InAb: A-0-0021.14 -RD- Axis is ready for power to the engine (Ab)
//   b_enable_FI_6: the enable of drive 6
//   b_enable_FI_5: the enable of drive 5
//   b_power_FI: close the polarization contactor
// label: (*power off FeedIndexer under panel mode*)
// fb_ton_powoff_FI(IN := NOT b_enable_FI AND b_local_on AND (axisdata[5].Axis_InAb OR axisdata[6].Axis_InAb), PT := T#2S); // TON
// b_enable_FI_6 R= fb_ton_powoff_FI.Q;
// b_enable_FI_5 R= fb_ton_powoff_FI.Q;
// b_power_FI R= fb_ton_powoff_FI.Q;

// NETWORK 31 (disabled)
//   b_SCC_enable_off: the command to disable all the drives
//   b_remote_on: in the remote mode
//   b_local_on: in the local mode
//   b_enable_az_1: the enable of drive 1
//   b_enable_az_2: the enable of drive 2
//   b_enable_el_3: the enable of drive 3
// label: (*the diasable command by TCP*)
// fb_ton_en_off(IN := b_SCC_enable_off AND (b_remote_on OR b_local_on), PT := t#5s); // TON
// rtrig_en_off(CLK := fb_ton_en_off.Q); // R_TRIG
// b_enable_az_1 R= rtrig_en_off.Q;
// b_enable_az_2 R= rtrig_en_off.Q;
// b_enable_el_3 R= rtrig_en_off.Q;

// NETWORK 32 (disabled)
//   axisdata[3].Axis_Power: A-0-0021.15 -RD- Axis has power on (AH_AF)
//   axisdata[2].Axis_Power: A-0-0021.15 -RD- Axis has power on (AH_AF)
//   axisdata[1].Axis_Power: A-0-0021.15 -RD- Axis has power on (AH_AF)
//   b_off_write: wrige cycle when it off
// fb_R_enable_off(CLK := NOT axisdata[3].Axis_Power AND NOT axisdata[2].Axis_Power AND NOT axisdata[1].Axis_Power); // R_TRIG
// b_off_write R= fb_R_enable_off.Q;

// NETWORK 33 (disabled)
//   b_lock_off: power off after arriving at the stow position
//   b_lock_off_m: power off after arriving at the maintain position
//   b_SCC_enable_off: the command to disable all the drives
//   b_remote_on: in the remote mode
//   b_local_on: in the local mode
//   axisdata[1].Axis_Error: A-0-0021.09 -RD- Axis reports error
//   axisdata[2].Axis_Error: A-0-0021.09 -RD- Axis reports error
//   axisdata[3].Axis_Error: A-0-0021.09 -RD- Axis reports error
//   FP_C_0_1030: Command: Clear all control errors
//   drive1: Real axis "Drive1" with axis number 1
// label: (*clear error if there is any error,when any disable command happens*)
// fb_ton_error(IN := b_lock_off OR b_lock_off_m OR b_SCC_enable_off AND (b_remote_on OR b_local_on), PT := t#5.5s); // TON
// FB_clear_all_error(
//     Execute := fb_ton_error.Q AND (axisdata[1].Axis_Error OR axisdata[2].Axis_Error OR axisdata[3].Axis_Error OR axisdata[7].Axis_Error OR axisdata[8].Axis_Error),
//     ParameterNumber := FP_C_0_1030,
//     Value := 3,
//     Axis := drive1); // MB_WriteParameter

// NETWORK 34
fb_blink_reset(ENABLE := lockstand, TIMELOW := t#100ms, TIMEHIGH := t#100ms); // BLINK
b_clear_error S= fb_blink_reset.OUT;

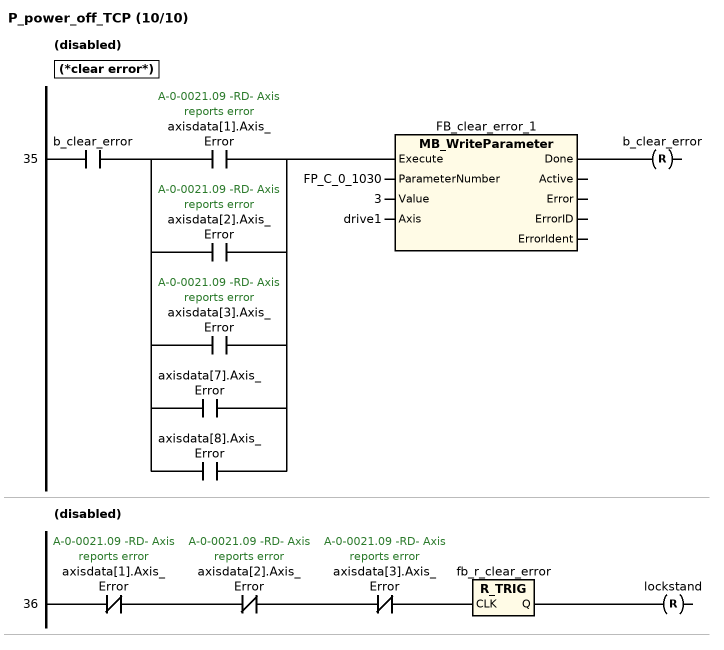
// NETWORK 35 (disabled)
//   axisdata[1].Axis_Error: A-0-0021.09 -RD- Axis reports error
//   axisdata[2].Axis_Error: A-0-0021.09 -RD- Axis reports error
//   axisdata[3].Axis_Error: A-0-0021.09 -RD- Axis reports error
//   FP_C_0_1030: Command: Clear all control errors
//   drive1: Real axis "Drive1" with axis number 1
// label: (*clear error*)
// FB_clear_error_1(
//     Execute := b_clear_error AND (axisdata[1].Axis_Error OR axisdata[2].Axis_Error OR axisdata[3].Axis_Error OR axisdata[7].Axis_Error OR axisdata[8].Axis_Error),
//     ParameterNumber := FP_C_0_1030,
//     Value := 3,
//     Axis := drive1); // MB_WriteParameter
// b_clear_error R= FB_clear_error_1.Done;

// NETWORK 36 (disabled)
//   axisdata[1].Axis_Error: A-0-0021.09 -RD- Axis reports error
//   axisdata[2].Axis_Error: A-0-0021.09 -RD- Axis reports error
//   axisdata[3].Axis_Error: A-0-0021.09 -RD- Axis reports error
// fb_r_clear_error(CLK := NOT axisdata[1].Axis_Error AND NOT axisdata[2].Axis_Error AND NOT axisdata[3].Axis_Error); // R_TRIG
// lockstand R= fb_r_clear_error.Q;

END_PROGRAM

// IndraMotionMlc1/Application/POUs/OPCUA/OPCUA_Node/P_Opcua_Azimuth
{attribute linkalways}
PROGRAM P_Opcua_Azimuth
VAR
	
END_VAR

Azimuth.Status.allActive:=(axisdata[1].Axis_Power AND axisdata[2].Axis_Power);
Azimuth.Status.Active:=b_PID_in_az;
Azimuth.Status.AxisMoving:=NOT(axisdata[1].rActualVelocity_i=0);;
IF status_code1 = 'F2042' OR status_code2 = 'F2042' THEN
	azimuth.Status.encBoxOp:=1;
ELSE
	azimuth.Status.encBoxOp:=0;
END_IF
azimuth.Status.EStop:=b_in_Estop;
IF status_code1 = 'F2028' OR status_code2 = 'F2028' THEN
	azimuth.Status.Exceed:=1;
ELSE
	azimuth.Status.Exceed:=0;
END_IF
azimuth.Status.InitOk:=axisdata[1].Axis_Inbb AND axisdata[1].Axis_Inbb;
azimuth.Status.LimOverride:=0;
IF status_code1 = 'F2037' OR status_code2 = 'F2037' THEN
	azimuth.Status.posDevOk:=1;
ELSE
	azimuth.Status.posDevOk:=0;
END_IF

Azimuth.Status.Reset:=0;
Azimuth.Status.SectorSw:=b_zone_az;
IF azimuth.Status.AxisState=axisStatetype.Standby THEN
	azimuth.Status.Ready:=1;
ELSE
	azimuth.Status.Ready:=0;
END_IF
//azimuth.Status.p_Act:=pointing.Status.TotalPointCorr_Az+r_pos_az;
//azimuth.Status.p_Enc:=r_pos_az;
azimuth.Status.p_PointCorr:=pointing.Status.TotalPointCorr_Az;

IF gc_b_sim_on THEN
	azimuth.Status.p_Set:=r_write_position_az_out;
END_IF

//azimuth.Status.p_Set:=P_shape_value[1];
//azimuth.Status.p_Shape:= P_shape_value[1];
//azimuth.Status.p_Shape:=r_write_position_az_out;

azimuth.Status.p_Dev:=Azimuth.Status.p_Set-Azimuth.Status.p_Enc;
azimuth.Status.v_Act:=axisdata[1].rActualVelocity_i*6;
azimuth.Status.v_Shape:=axisdata[1].rActualVelocity_i*6;
azimuth.Status.v_SetMax:=r_vel_max_Az*6;
(***************AxisState**************)


IF (axisdata[1].Axis_Inbb AND axisdata[2].Axis_Inbb) THEN
	Azimuth.Status.AxisState:=axisstatetype.StartUp;
END_IF
IF (axisdata[1].Axis_InAb AND axisdata[2].Axis_InAb) THEN
	Azimuth.Status.AxisState:=axisstatetype.Standby;
END_IF

IF  b_stow_pin_limit_lock THEN
	Azimuth.Status.AxisState:=axisstatetype.Stowed;	
END_IF

IF  b_scc_enable_on OR b_activate_Az THEN
	azimuth.Status.AxisState:=AxisStateType.Activating;
END_IF

IF  b_scc_enable_off OR b_deactivate_Az THEN
	azimuth.Status.AxisState:=AxisStateType.Deactivating;
END_IF

IF b_PID_in_az THEN
	azimuth.Status.AxisState:=AxisStateType.Standstill;
END_IF

IF  b_track_on AND (ABS(axisdata[1].rActualVelocity_i) < (gc_r_vel_tracking_limit_Az-0.001)) THEN
	azimuth.Status.AxisState:=AxisStateType.Track;
END_IF

IF b_Estop_active OR b_interlock_active_Az THEN
	azimuth.Status.AxisState:=AxisStateType.Locked;
END_IF

IF (b_Estop_active OR b_interlock_active_Az) AND b_stow_pin_limit_lock  THEN
	azimuth.Status.AxisState:=AxisStateType.Locked_Stowed;
END_IF

IF axisdata[1].Stopping THEN
	azimuth.Status.AxisState:=AxisStateType.Stopping;
END_IF

IF (ABS(axisdata[1].rActualVelocity_i) > (gc_r_vel_tracking_limit_Az+0.001)) OR axisdata[7].DiscreteMotion THEN
	azimuth.Status.AxisState:=AxisStateType.Slew;
END_IF
(**********axis status end***********)

// Axis Statemachine attempt
(*
CASE Azimuth.Status.AxisState OF
	AxisStatetype.Activating:
       IF b_PID_in_az THEN // exit condition 
       		Azimuth.Status.AxisState:=AxisStatetype.Standstill;
       END_IF
	AxisStatetype.Deactivating:
	  IF b_power_az = False Then 
	     Azimuth.Status.AxisState:=AxisStatetype.Standby;
      End_IF
	AxisStatetype.Jog:
	  IF b_local_on AND NOT(Azimuth.Status.AxisMoving) THEN 
		 Azimuth.Status.AxisState:=AxisStateType.Standstill;
	  END_IF
	AxisStatetype.Locked:
	   IF NOT(b_interlock_active_Az) THEN
		   Azimuth.Status.AxisState:=AxisStateType.Standby;
	   END_IF
	AxisStatetype.Locked_Stowed:
	   IF NOT(b_interlock_active_Az) AND NOT(b_Estop_active) THEN
		   Azimuth.Status.AxisState:=AxisStateType.Stowed;
	   END_IF
	AxisStatetype.Slew:
         IF b_track_on AND Management.Status.OnSource THEN
           Azimuth.Status.AxisState:=AxisStateType.Track;
		 ELSIF b_stop_Az OR b_deactivate_Az OR b_Estop_active THEN
			  Azimuth.Status.AxisState:=AxisStateType.Stopping;
		 END_IF
			 
	AxisStatetype.Standby:
         IF b_enable_Az OR b_activate_Az THEN 
  			Azimuth.Status.AxisState:=AxisStateType.Activating;
		 END_IF
	AxisStatetype.Standstill:
	    IF b_local_on AND Azimuth.Status.AxisMoving THEN 
			Azimuth.Status.AxisState:=AxisStatetype.Jog;
		ELSIF b_track_on THEN 
			Azimuth.Status.AxisState:=AxisStatetype.Track;
		ELSIF b_moving_Az THEN
	        Azimuth.Status.AxisState:=AxisStatetype.Slew;
		ELSIF b_deactivate_Az THEN 
			Azimuth.Status.AxisState:=AxisStatetype.Deactivating;
		END_IF
	AxisStatetype.StartUp:
		IF (axisdata[1].Axis_InAb AND axisdata[2].Axis_InAb) THEN
			Azimuth.Status.AxisState:=axisstatetype.Standby;
        END_IF					
	AxisStatetype.Stopping:
		IF NOT(Azimuth.Status.AxisMoving) THEN
		   Azimuth.Status.AxisState:=AxisStateType.Standstill;
		END_IF
	AxisStatetype.Stowed:
		IF b_stow_pin_limit_unlock THEN
			Azimuth.Status.AxisState:=axisstatetype.Standby;
        END_IF		
	AxisStatetype.Track:
          IF NOT b_track_on THEN 
			Azimuth.Status.AxisState:=AxisStateType.Stopping;
		  ELSIF (axisdata[1].rActualVelocity_i > r_vel_tracking_limit_Az) THEN
			Azimuth.Status.AxisState:=AxisStateType.Slew;
		  ELSIF b_stop_Az OR b_deactivate_Az THEN
			  Azimuth.Status.AxisState:=AxisStateType.Stopping;
		 END_IF
	
			  
END_CASE
*)




(******ErrorStatus******)
IF axisdata[1].Axis_Error OR axisdata[2].Axis_Error THEN
	azimuth.ErrorStatus.errErrorActive:=1;
ELSE
	azimuth.ErrorStatus.errErrorActive:=0;
END_IF
azimuth.ErrorStatus.errFieldBus:=0;
azimuth.ErrorStatus.errLim2CCW:=b_limit_final_ccw_az;
azimuth.ErrorStatus.errLim2CW:=b_limit_final_cw_az;
IF status_code1 = 'E2059' OR status_code2 = 'E2059' THEN
	azimuth.ErrorStatus.errLimV_Err:=1;
ELSE
	azimuth.ErrorStatus.errLimV_Err:=0;
END_IF
azimuth.ErrorStatus.errMotComm:=(axisdata[1].Axis_NRT OR axisdata[2].Axis_NRT);
IF status_code1 = 'F2031' OR status_code2 = 'F2031' THEN
	azimuth.ErrorStatus.errMotEnc:=1;
ELSE
	azimuth.ErrorStatus.errMotEnc:=0;
END_IF
IF status_code1 = 'F2021' OR status_code2 = 'F2021' OR azimuth.ErrorStatus.errMotEnc THEN
	azimuth.ErrorStatus.errMotor:=1;
ELSE
	azimuth.ErrorStatus.errMotor:=0;
END_IF
IF azimuth.ErrorStatus.errMotor OR azimuth.ErrorStatus.errMotEnc THEN
	azimuth.ErrorStatus.errMotReady:=1;
ELSE
	azimuth.ErrorStatus.errMotReady:=0;
END_IF
azimuth.ErrorStatus.errOverride:=0;
azimuth.ErrorStatus.errV_DevExceed:=azimuth.ErrorStatus.errLimV_Err;
IF status_code1 = 'F2075' THEN
	azimuth.ErrorStatus.errP_RangeExceed:=1;
ELSE
	azimuth.ErrorStatus.errP_RangeExceed:=0;
END_IF
IF status_code1 = 'F2037' OR status_code2 = 'F2037' THEN
	azimuth.ErrorStatus.errP_DevExceed:=1;
ELSE
	azimuth.ErrorStatus.errP_DevExceed:=0;
END_IF
azimuth.ErrorStatus.errPosEnc:=azimuth.Status.encBoxOp;
azimuth.ErrorStatus.errPosEnc_Fo:=azimuth.Status.encBoxOp;
IF status_code1 = 'F2026' OR status_code2 = 'F2026' THEN
	azimuth.ErrorStatus.errPower:=1;
ELSE
	azimuth.ErrorStatus.errPower:=0;
END_IF
(***** Error status end*****)


(*******Warning state********)
azimuth.WarningStatus.waLim1CW:=b_limit_cw_az;
azimuth.WarningStatus.waLim1CCW:=b_limit_ccw_az;
IF status_code1 = 'E8029' OR status_code2 = 'E8029' THEN
	azimuth.WarningStatus.waLimSoftCW:=1;
ELSE
	azimuth.WarningStatus.waLimSoftCW:=0;
END_IF
IF status_code1 = 'E8030' OR status_code2 = 'E8030' THEN
	azimuth.WarningStatus.waLimSoftCCW:=1;
ELSE
	azimuth.WarningStatus.waLimSoftCCW:=0;
END_IF
IF status_code1 = 'E8260' OR status_code2 = 'E8260' THEN
	azimuth.WarningStatus.waMmaxExceeded:=1;
ELSE
	azimuth.WarningStatus.waMmaxExceeded:=0;
END_IF
azimuth.WarningStatus.waMotReady:=azimuth.ErrorStatus.errMotReady;
azimuth.WarningStatus.waMotWarn:=(axisdata[1].Axis_Warning OR axisdata[1].Axis_Warning);
azimuth.WarningStatus.waOverride:=0;
azimuth.WarningStatus.waParamFault:=(azimuth.WarningStatus.waMotReady OR azimuth.ErrorStatus.errMotReady);
IF status_code1 = 'E2031' OR status_code2 = 'E2031' THEN
	azimuth.WarningStatus.waPosEncWarn:=1;
ELSE
	azimuth.WarningStatus.waPosEncWarn:=0;
END_IF
azimuth.WarningStatus.waStowPinsDep:=b_stow_pin_limit_lock;
azimuth.WarningStatus.waVelLimit:=azimuth.ErrorStatus.errV_DevExceed;
(*********Warning status end***********)
(*****motor1****)
azimuth.MotorOne.ErrorCode:= STRING_TO_UINT(status_code1);
azimuth.MotorOne.mActTorq:=r_torque_1*60.5;
azimuth.MotorOne.mActVelocity:=i_speed_1;
azimuth.MotorOne.MotorTemp:=r_temp_motor1;
azimuth.MotorOne.RateOfUtil:=r_torque_1;
azimuth.MotorOne.MotorOverload:=r_torque_1;
(*****motor2****)
azimuth.MotorTwo.ErrorCode:= STRING_TO_UINT(status_code2);
azimuth.MotorTwo.mActTorq:=r_torque_2*60.5;
azimuth.MotorTwo.mActVelocity:=i_speed_2;
azimuth.MotorTwo.MotorTemp:=r_temp_motor2;
azimuth.MotorTwo.RateOfUtil:=r_torque_2;
azimuth.MotorTwo.MotorOverload:=r_torque_2;

END_PROGRAM

// IndraMotionMlc1/Application/POUs/OPCUA/OPCUA_Node/P_Opcua_Elevation
PROGRAM P_Opcua_Elevation
VAR
	
END_VAR

Elevation.Status.AllActive:=axisdata[3].Axis_Power;
Elevation.Status.Active:=axisdata[3].Axis_InSynchron;
Elevation.Status.AxisMoving:=NOT(axisdata[3].rActualVelocity_i=0);
IF status_code3 = 'F2042' OR status_code4 = 'F2042' THEN
	Elevation.Status.encBoxOp:=1;
ELSE
	Elevation.Status.encBoxOp:=0;
END_IF
Elevation.Status.EStop:=b_in_Estop;
IF status_code3 = 'F2028'THEN
	Elevation.Status.Exceed:=1;
ELSE
	Elevation.Status.Exceed:=0;
END_IF
Elevation.Status.InitOk:=axisdata[3].Axis_Inbb;
Elevation.Status.LimOverride:=0;
IF status_code3 = 'F2037' THEN
	Elevation.Status.posDevOk:=1;
ELSE
	Elevation.Status.posDevOk:=0;
END_IF

Elevation.Status.Reset:=0;
Elevation.Status.SectorSw:=b_zone_az;
IF Elevation.Status.AxisState=axisStatetype.Standby THEN
	Elevation.Status.Ready:=1;
ELSE
	Elevation.Status.Ready:=0;
END_IF
//Elevation.Status.p_Act:=pointing.Status.TotalPointCorr_El+r_pos_el;
//Elevation.Status.p_Enc:=r_pos_el;
Elevation.Status.p_PointCorr:=pointing.Status.TotalPointCorr_El;
IF gc_b_sim_on THEN
	Elevation.Status.p_Set:=r_write_position_el_out;
END_IF

//Elevation.Status.p_Set:=P_shape_value[3];
//Elevation.Status.p_Shape:= P_shape_value[3];
Elevation.Status.p_Shape:=r_write_position_el_out;
Elevation.Status.p_Dev:=Elevation.Status.p_Shape-Elevation.Status.p_Enc;
Elevation.Status.v_Act:=axisdata[3].rActualVelocity_i*6;
Elevation.Status.v_Shape:=axisdata[3].rActualVelocity_i*6;
Elevation.Status.v_SetMax:= r_vel_max_El*6;
//Elevation.Status.v_Act:=V_act_value[3];
//Elevation.Status.v_Shape:=V_shape_value[3];


(***************AxisState**************)

IF axisdata[3].Axis_Inbb  THEN
	Elevation.Status.AxisState:=axisstatetype.StartUp;
END_IF
IF axisdata[3].Axis_InAb  THEN
	Elevation.Status.AxisState:=axisstatetype.Standby;
END_IF

IF  b_stow_pin_limit_lock THEN
	Elevation.Status.AxisState:=axisstatetype.Stowed;	
END_IF

IF  b_scc_enable_on OR b_activate_El THEN
	Elevation.Status.AxisState:=AxisStateType.Activating;
END_IF

IF  b_scc_enable_off OR b_deactivate_El THEN
	Elevation.Status.AxisState:=AxisStateType.Deactivating;
END_IF

IF b_PID_in_El THEN
	Elevation.Status.AxisState:=AxisStateType.Standstill;
END_IF

IF  b_track_on AND (ABS(axisdata[3].rActualVelocity_i) < gc_r_vel_tracking_limit_El) THEN
	Elevation.Status.AxisState:=AxisStateType.Track;
END_IF

IF b_Estop_active OR b_interlock_active_El THEN
	Elevation.Status.AxisState:=AxisStateType.Locked;
END_IF

IF (b_Estop_active OR b_interlock_active_El) AND b_stow_pin_limit_lock  THEN
	Elevation.Status.AxisState:=AxisStateType.Locked_Stowed;
END_IF

IF axisdata[3].Stopping THEN
	Elevation.Status.AxisState:=AxisStateType.Stopping;
END_IF

IF (ABS(axisdata[3].rActualVelocity_i) > gc_r_vel_tracking_limit_El) OR axisdata[8].DiscreteMotion THEN
	Elevation.Status.AxisState:=AxisStateType.Slew;
END_IF
(**********axis status end***********)


(******ErrorStatus******)
IF axisdata[3].Axis_Error THEN
	Elevation.ErrorStatus.errErrorActive:=1;
ELSE
	Elevation.ErrorStatus.errErrorActive:=0;
END_IF
Elevation.ErrorStatus.errFieldBus:=0;
Elevation.ErrorStatus.errLim2CCW:=b_limit_final_ccw_el;
Elevation.ErrorStatus.errLim2CW:=b_limit_final_cw_el;
IF status_code3 = 'E2059' THEN
	Elevation.ErrorStatus.errLimV_Err:=1;
ELSE
	Elevation.ErrorStatus.errLimV_Err:=0;
END_IF
Elevation.ErrorStatus.errMotComm:=(axisdata[3].Axis_NRT OR axisdata[2].Axis_NRT);
IF status_code3 = 'F2031' THEN
	Elevation.ErrorStatus.errMotEnc:=1;
ELSE
	Elevation.ErrorStatus.errMotEnc:=0;
END_IF
IF status_code3 = 'F2021' OR Elevation.ErrorStatus.errMotEnc THEN
	Elevation.ErrorStatus.errMotor:=1;
ELSE
	Elevation.ErrorStatus.errMotor:=0;
END_IF
IF Elevation.ErrorStatus.errMotor OR Elevation.ErrorStatus.errMotEnc THEN
	Elevation.ErrorStatus.errMotReady:=1;
ELSE
	Elevation.ErrorStatus.errMotReady:=0;
END_IF
Elevation.ErrorStatus.errOverride:=0;
Elevation.ErrorStatus.errV_DevExceed:=Elevation.ErrorStatus.errLimV_Err;
IF status_code3 = 'F2075' THEN
	Elevation.ErrorStatus.errP_RangeExceed:=1;
ELSE
	Elevation.ErrorStatus.errP_RangeExceed:=0;
END_IF
IF status_code3 = 'F2037' THEN
	Elevation.ErrorStatus.errP_DevExceed:=1;
ELSE
	Elevation.ErrorStatus.errP_DevExceed:=0;
END_IF
Elevation.ErrorStatus.errPosEnc:=Elevation.Status.encBoxOp;
Elevation.ErrorStatus.errPosEnc_Fo:=Elevation.Status.encBoxOp;
IF status_code3 = 'F2026' THEN
	Elevation.ErrorStatus.errPower:=1;
ELSE
	Elevation.ErrorStatus.errPower:=0;
END_IF
(***** Error status end*****)


(*******Warning state********)
Elevation.WarningStatus.waLim1CW:=b_limit_cw_el;
Elevation.WarningStatus.waLim1CCW:=b_limit_ccw_el;
IF status_code3 = 'E8029' THEN
	Elevation.WarningStatus.waLimSoftCW:=1;
ELSE
	Elevation.WarningStatus.waLimSoftCW:=0;
END_IF
IF status_code3 = 'E8030'  THEN
	Elevation.WarningStatus.waLimSoftCCW:=1;
ELSE
	Elevation.WarningStatus.waLimSoftCCW:=0;
END_IF
IF status_code3 = 'E8260' THEN
	Elevation.WarningStatus.waMmaxExceeded:=1;
ELSE
	Elevation.WarningStatus.waMmaxExceeded:=0;
END_IF
Elevation.WarningStatus.waMotReady:=Elevation.ErrorStatus.errMotReady;
Elevation.WarningStatus.waMotWarn:=axisdata[3].Axis_Warning;
Elevation.WarningStatus.waOverride:=0;
Elevation.WarningStatus.waParamFault:=Elevation.WarningStatus.waMotReady;
IF status_code3 = 'E2031' THEN
	Elevation.WarningStatus.waPosEncWarn:=1;
ELSE
	Elevation.WarningStatus.waPosEncWarn:=0;
END_IF
//Elevation.WarningStatus.waStowPinsDep:=b_limit_lock;
Elevation.WarningStatus.waVelLimit:=Elevation.ErrorStatus.errV_DevExceed;
(*********Warning status end***********)
(*****motor1****)
Elevation.MotorOne.ErrorCode:= STRING_TO_UINT(status_code3);
Elevation.MotorOne.mActTorq:=r_torque_3*82.5;
Elevation.MotorOne.mActVelocity:=i_speed_3;
Elevation.MotorOne.MotorTemp:=r_temp_motor3;
Elevation.MotorOne.RateOfUtil:=r_torque_3;
Elevation.MotorOne.MotorOverload:=r_torque_3;
(*****motor2****)
(*Elevation.MotorTwo.ErrorCode:= STRING_TO_DINT(status_code2);
Elevation.MotorTwo.mActTorq:=r_torque_2*60.5;
Elevation.MotorTwo.mActVelocity:=i_speed_2;
Elevation.MotorTwo.MotorTemp:=r_temp_motor2;
Elevation.MotorTwo.RateOfUtil:=r_torque_2;
Elevation.MotorTwo.MotorOverload:=r_torque_2;
*)

END_PROGRAM

// IndraMotionMlc1/Application/POUs/OPCUA/OPCUA_Node/P_Opcua_FeedIndexer
PROGRAM P_Opcua_FeedIndexer
VAR
END_VAR

FeedIndexer.Status.allActive:=(axisdata[5].Axis_Power AND axisdata[6].Axis_Power);
FeedIndexer.Status.Active:=b_PID_in_FI;
FeedIndexer.Status.AxisMoving:=NOT(axisdata[5].rActualVelocity_i=0);
IF status_code4 = 'F2042' OR status_code5 = 'F2042' THEN
	FeedIndexer.Status.encBoxOp:=1;
ELSE
	FeedIndexer.Status.encBoxOp:=0;
END_IF
FeedIndexer.Status.EStop:=b_in_Estop;
IF status_code4 = 'F2028' OR status_code5 = 'F2028' THEN
	FeedIndexer.Status.Exceed:=1;
ELSE
	FeedIndexer.Status.Exceed:=0;
END_IF
FeedIndexer.Status.InitOk:=axisdata[5].Axis_Inbb AND axisdata[6].Axis_Inbb;
FeedIndexer.Status.LimOverride:=0;
IF status_code4 = 'F2037' OR status_code5 = 'F2037' THEN
	FeedIndexer.Status.posDevOk:=1;
ELSE
	FeedIndexer.Status.posDevOk:=0;
END_IF

FeedIndexer.Status.Reset:=0;
//FeedIndexer.SectorSw:=b_zone_FI;
IF FeedIndexer.Status.AxisState=axisStatetype.Standby THEN
	FeedIndexer.Status.Ready:=1;
ELSE
	FeedIndexer.Status.Ready:=0;
END_IF
FeedIndexer.Status.p_Act:=r_pos_FI; 
FeedIndexer.Status.p_Enc:=r_pos_FI;
FeedIndexer.Status.p_PointCorr:=0;


//FeedIndexer.Status.p_Set:=r_write_position_fi_out;
//FeedIndexer.Status.p_Shape:= P_shape_value[4];
//FeedIndexer.Status.p_Set:=r_write_position_fi_out;
FeedIndexer.Status.p_Shape:=r_write_position_fi_out;;
FeedIndexer.Status.p_Dev:=FeedIndexer.Status.p_Set-FeedIndexer.Status.p_Enc;
//FeedIndexer.Status.v_Act:=V_act_value[4];
//FeedIndexer.Status.v_Shape:=V_shape_value[4];
FeedIndexer.Status.v_Act:=axisdata[9].rActualVelocity_i*6;
FeedIndexer.Status.v_Shape:=axisdata[9].rActualVelocity_i*6;
FeedIndexer.Status.v_SetMax:=r_vel_max_Fi*6;

	


(***************AxisState**************)
IF (axisdata[4].Axis_Inbb AND axisdata[5].Axis_Inbb) THEN
	FeedIndexer.Status.AxisState:=AxisStateType.StartUp;
END_IF
IF (axisdata[4].Axis_InAb AND axisdata[5].Axis_InAb) THEN
	FeedIndexer.Status.AxisState:=AxisStateType.Standby;
END_IF

IF  b_scc_enable_on OR b_activate_FI THEN
	FeedIndexer.Status.AxisState:=AxisStateType.Activating;
END_IF

IF  b_scc_enable_off OR b_deactivate_FI THEN
	FeedIndexer.Status.AxisState:=AxisStateType.Deactivating;
END_IF

IF b_PID_in_FI THEN
	FeedIndexer.Status.AxisState:=AxisStateType.Standstill;
END_IF


(*IF  b_track_on  THEN
	FeedIndexer.Status.AxisState:=AxisStateType.Track;
END_IF *)

IF b_Estop_active and b_interlock_active_Fi THEN
	FeedIndexer.Status.AxisState:=AxisStateType.Locked;
END_IF
IF axisdata[9].Stopping  THEN
	FeedIndexer.Status.AxisState:=AxisStateType.Stopping;
END_IF

IF ABS(axisdata[9].rActualVelocity_i) > gc_r_vel_tracking_limit_Fi THEN
	FeedIndexer.Status.AxisState:=AxisStateType.Slew;
END_IF
(**********axis status end***********)


(******ErrorStatus******)
IF axisdata[4].Axis_Error OR axisdata[5].Axis_Error THEN
	FeedIndexer.ErrorStatus.errErrorActive:=1;
ELSE
	FeedIndexer.ErrorStatus.errErrorActive:=0;
END_IF
FeedIndexer.ErrorStatus.errFieldBus:=0;
FeedIndexer.ErrorStatus.errLim2CCW:=b_limit_final_ccw_FI;
FeedIndexer.ErrorStatus.errLim2CW:=b_limit_final_cw_FI;
IF status_code4 = 'E2059' OR status_code5 = 'E2059' THEN
	FeedIndexer.ErrorStatus.errLimV_Err:=1;
ELSE
	FeedIndexer.ErrorStatus.errLimV_Err:=0;
END_IF
FeedIndexer.ErrorStatus.errMotComm:=(axisdata[5].Axis_NRT OR axisdata[6].Axis_NRT);
IF status_code4 = 'F2031' OR status_code5 = 'F2031' THEN
	FeedIndexer.ErrorStatus.errMotEnc:=1;
ELSE
	FeedIndexer.ErrorStatus.errMotEnc:=0;
END_IF
IF status_code4 = 'F2021' OR status_code5 = 'F2021' OR FeedIndexer.ErrorStatus.errMotEnc THEN
	FeedIndexer.ErrorStatus.errMotor:=1;
ELSE
	FeedIndexer.ErrorStatus.errMotor:=0;
END_IF
IF FeedIndexer.ErrorStatus.errMotor OR FeedIndexer.ErrorStatus.errMotEnc THEN
	FeedIndexer.ErrorStatus.errMotReady:=1;
ELSE
	FeedIndexer.ErrorStatus.errMotReady:=0;
END_IF
FeedIndexer.ErrorStatus.errOverride:=0;
FeedIndexer.ErrorStatus.errV_DevExceed:=FeedIndexer.ErrorStatus.errLimV_Err;
IF status_code4 = 'F2075' THEN
	FeedIndexer.ErrorStatus.errP_RangeExceed:=1;
ELSE
	FeedIndexer.ErrorStatus.errP_RangeExceed:=0;
END_IF
IF status_code4 = 'F2037' OR status_code5 = 'F2037' THEN
	FeedIndexer.ErrorStatus.errP_DevExceed:=1;
ELSE
	FeedIndexer.ErrorStatus.errP_DevExceed:=0;
END_IF
FeedIndexer.ErrorStatus.errPosEnc:=FeedIndexer.Status.encBoxOp;
FeedIndexer.ErrorStatus.errPosEnc_Fo:=FeedIndexer.Status.encBoxOp;
IF status_code4 = 'F2026' OR status_code5 = 'F2026' THEN
	FeedIndexer.ErrorStatus.errPower:=1;
ELSE
	FeedIndexer.ErrorStatus.errPower:=0;
END_IF
(***** Error status end*****)


(*******Warning state********)
FeedIndexer.WarningStatus.waLim1CW:=b_limit_cw_FI;
FeedIndexer.WarningStatus.waLim1CCW:=b_limit_ccw_FI;
IF status_code4 = 'E8029' OR status_code5 = 'E8029' THEN
	FeedIndexer.WarningStatus.waLimSoftCW:=1;
ELSE
	FeedIndexer.WarningStatus.waLimSoftCW:=0;
END_IF
IF status_code4 = 'E8030' OR status_code5 = 'E8030' THEN
	FeedIndexer.WarningStatus.waLimSoftCCW:=1;
ELSE
	FeedIndexer.WarningStatus.waLimSoftCCW:=0;
END_IF
IF status_code4 = 'E8260' OR status_code5 = 'E8260' THEN
	FeedIndexer.WarningStatus.waMmaxExceeded:=1;
ELSE
	FeedIndexer.WarningStatus.waMmaxExceeded:=0;
END_IF
FeedIndexer.WarningStatus.waMotReady:=FeedIndexer.ErrorStatus.errMotReady;
FeedIndexer.WarningStatus.waMotWarn:=(axisdata[4].Axis_Warning OR axisdata[4].Axis_Warning);
FeedIndexer.WarningStatus.waOverride:=0;
FeedIndexer.WarningStatus.waParamFault:=(FeedIndexer.WarningStatus.waMotReady OR FeedIndexer.ErrorStatus.errMotReady);
IF status_code4 = 'E2031' OR status_code5 = 'E2031' THEN
	FeedIndexer.WarningStatus.waPosEncWarn:=1;
ELSE
	FeedIndexer.WarningStatus.waPosEncWarn:=0;
END_IF
FeedIndexer.WarningStatus.waStowPinsDep:=FALSE;
FeedIndexer.WarningStatus.waVelLimit:=FeedIndexer.ErrorStatus.errV_DevExceed;
(*********Warning status end***********)
(*****motor1****)
FeedIndexer.MotorOne.ErrorCode:= STRING_TO_UINT(status_code4);
FeedIndexer.MotorOne.mActTorq:=r_torque_4*7.1;
FeedIndexer.MotorOne.mActVelocity:=i_speed_4;
FeedIndexer.MotorOne.MotorTemp:=r_temp_motor4;
FeedIndexer.MotorOne.RateOfUtil:=r_torque_4;
FeedIndexer.MotorOne.MotorOverload:=r_torque_4;
(*****motor2****)
FeedIndexer.MotorTwo.ErrorCode:= STRING_TO_UINT(status_code5);
FeedIndexer.MotorTwo.mActTorq:=r_torque_5*7.1;
FeedIndexer.MotorTwo.mActVelocity:=i_speed_5;
FeedIndexer.MotorTwo.MotorTemp:=r_temp_motor5;
FeedIndexer.MotorTwo.RateOfUtil:=r_torque_5;
FeedIndexer.MotorTwo.MotorOverload:=r_torque_5;

END_PROGRAM

// IndraMotionMlc1/Application/POUs/OPCUA/OPCUA_Node/P_Opcua_Safety
PROGRAM P_Opcua_Safety
VAR
	b_final_limit_active:BOOL;
	fb_move_stow_Az: MC_MoveAbsolute;
	fb_move_stow_El: MC_MoveAbsolute;
	fb_ton_stow: TON;
	fb_self_reset_stow: R_Trig;
	fb_ton_self_reset_stow: TON;
	fb_rtrig_off_stow:R_Trig;
	fb_rtrig_lock_stow: R_Trig;
	fb_rtrig_reset_deploy: R_Trig;
	fb_rtrig_reset_retract: R_Trig;
	fb_rtrig_estop: R_TRIG;
	fb_rtrig_interlock_Az: R_TRIG;
	fb_rtrig_interlock_El: R_TRIG;
	fb_rtrig_interlock_Fi: R_TRIG;
	
	fb_ton_sim_stow: TON;
	_retract: TON;
	fb_ton_sim_retract: TON;
	fb_ton_sim_deploy: TON;
	fb_rtrig_sim_retract: R_TRIG;
	fb_rtrig_sim_deploy: R_TRIG;
	fb_rtrig_stow_deactivate: R_TRIG;
	fb_rtrig_stow_pulse: R_TRIG;
	_test: BOOL;
	b_stow_SIP: BOOL;
	rtrig_Estop_Az: R_TRIG;
	fb_Estop_Az: MC_Stop;
	rtrig_Estop_El: R_TRIG;
	fb_Estop_El: MC_Stop;
	rtrig_Estop_Fi: R_TRIG;
	fb_Estop_Fi: MC_Stop;
	MC_MoveRelative_0: MC_MoveRelative;
	MC_MoveRelative_1: MC_MoveRelative;
	R_TRIG_0: R_TRIG;
	TON_0: TON;
	b_stow_wait: BOOL;
	TON_1: TON;
	b_stow_run: BOOL;
	R_TRIG_1: R_TRIG;
	F_TRIG_0: F_TRIG;
	F_TRIG_1: F_TRIG;
	F_TRIG_2: F_TRIG;
	F_TRIG_3: F_TRIG;
	F_TRIG_4: F_TRIG;
END_VAR
VAR // added by the converter: edge detectors and wires of the graphical bodies
    _w1, _w2, _w3, _w4, _w5 : BOOL;
END_VAR

safety();
(*IF b_HHP_Estop OR b_Turnhead_Estop OR b_DS_Estop OR b_FI_Estop OR b_Turnhead_Hatch OR b_AZ_Hatch OR (NOT(b_stow_pin_limit_unlock)) THEN
	b_in_interlock:=1;
ELSE
	b_in_interlock:=0;
END_IF*)

(*IF b_in_interlock OR b_DSDoor_Estop OR b_PSCDoor_Estop OR b_DriveCabinetDoor_Estop OR b_EMISCDoor_Estop THEN // b_in_interlock true will cause an EStop. Whereas it should only cause an interlock. 
	b_in_Estop:=1;
ELSE
	b_in_Estop:=0;
END_IF*)
safety.Status.AutoStowActive:=0;
safety.Status.Axes_InitFault:=NOT(Azimuth.Status.InitOk AND Elevation.Status.InitOk AND FeedIndexer.Status.InitOk);
safety.Status.EStopFi:=b_FI_Estop;
safety.Status.EStopHHP:=b_HHP_Estop;
safety.Status.EStopPED:=b_DS_Estop;
safety.Status.EStopTurnhead:=b_Turnhead_Estop;
safety.Status.HatchTurnheadRoof:=b_Turnhead_Hatch;
safety.Status.HatchAzBearing:=b_AZ_Hatch;
//safety.InterlockAck
safety.Status.Lim2_CCW_Az:=b_limit_final_ccw_az;
safety.Status.Lim2_CCW_Fi:=b_limit_final_ccw_Fi;
safety.Status.Lim2_CW_Az:=b_limit_final_cw_az;
safety.Status.Lim2_CW_Fi:=b_limit_final_cw_Fi;
safety.Status.Lim2_Dn_El:=b_limit_final_ccw_el;
safety.Status.Lim2_Up_El:=b_limit_final_cw_el;
b_final_limit_active:=(safety.Status.Lim2_CCW_Az OR safety.Status.Lim2_CW_Az OR safety.Status.Lim2_Dn_El OR safety.Status.Lim2_Up_El OR safety.Status.Lim2_CCW_Fi OR safety.Status.Lim2_CW_Fi); 

(* Still to be wired in *)
safety.Status.SafetyLockout_Az:=b_Lock_Out_Az;
safety.Status.SafetyLockout_El:=b_Lock_Out_El;
safety.Status.SafetyLockout_Fi:=b_Lock_Out_Fi;

IF safety.Status.Axes_InitFault THEN
	safety.Status.SafetyState:=SafetyStatetype.Stopped;
ELSIF b_in_interlock OR b_in_Estop OR b_final_limit_active THEN
	safety.Status.SafetyState:=SafetyStatetype.Error;
ELSE
	safety.Status.SafetyState:=SafetyStatetype.Running;	
END_IF
safety.Status.STO_Az:=b_in_interlock;
safety.Status.STO_El:=b_in_interlock;
safety.Status.STO_Fi:=b_in_interlock;

IF b_stow_pin_deploy THEN
	safety.Status.StowPinStatus:=StowPinStatustype.Deploying;
ELSIF b_stow_pin_limit_lock THEN
	safety.Status.StowPinStatus:=StowPinStatustype.Deployed;
ELSIF b_stow_pin_retract AND NOT(b_stow_pin_limit_unlock) THEN
	safety.Status.StowPinStatus:=StowPinStatustype.Retracting;
ELSIF b_stow_pin_limit_unlock THEN
	safety.Status.StowPinStatus:=StowPinStatustype.Retracted;
END_IF

IF (Azimuth.Status.p_Enc >= Azimuth.Status.StowPos_Minus AND Azimuth.Status.p_Enc <= Azimuth.Status.StowPos_Plus) THEN
	b_stow_lock_allow:=1;
ELSE 
	b_stow_lock_allow:=0;
END_IF

(*
IF b_in_interlock AND b_in_Estop THEN 
	Safety.Status.InterlockClearable:=0;
ELSE
	Safety.Status.InterlockClearable:=1;	
END_IF *)

// Run Ladder Logic
P_Opcua_Safety.A_STOW();
P_Opcua_Safety.A_Interlock_Estop();

ACTION A_STOW:
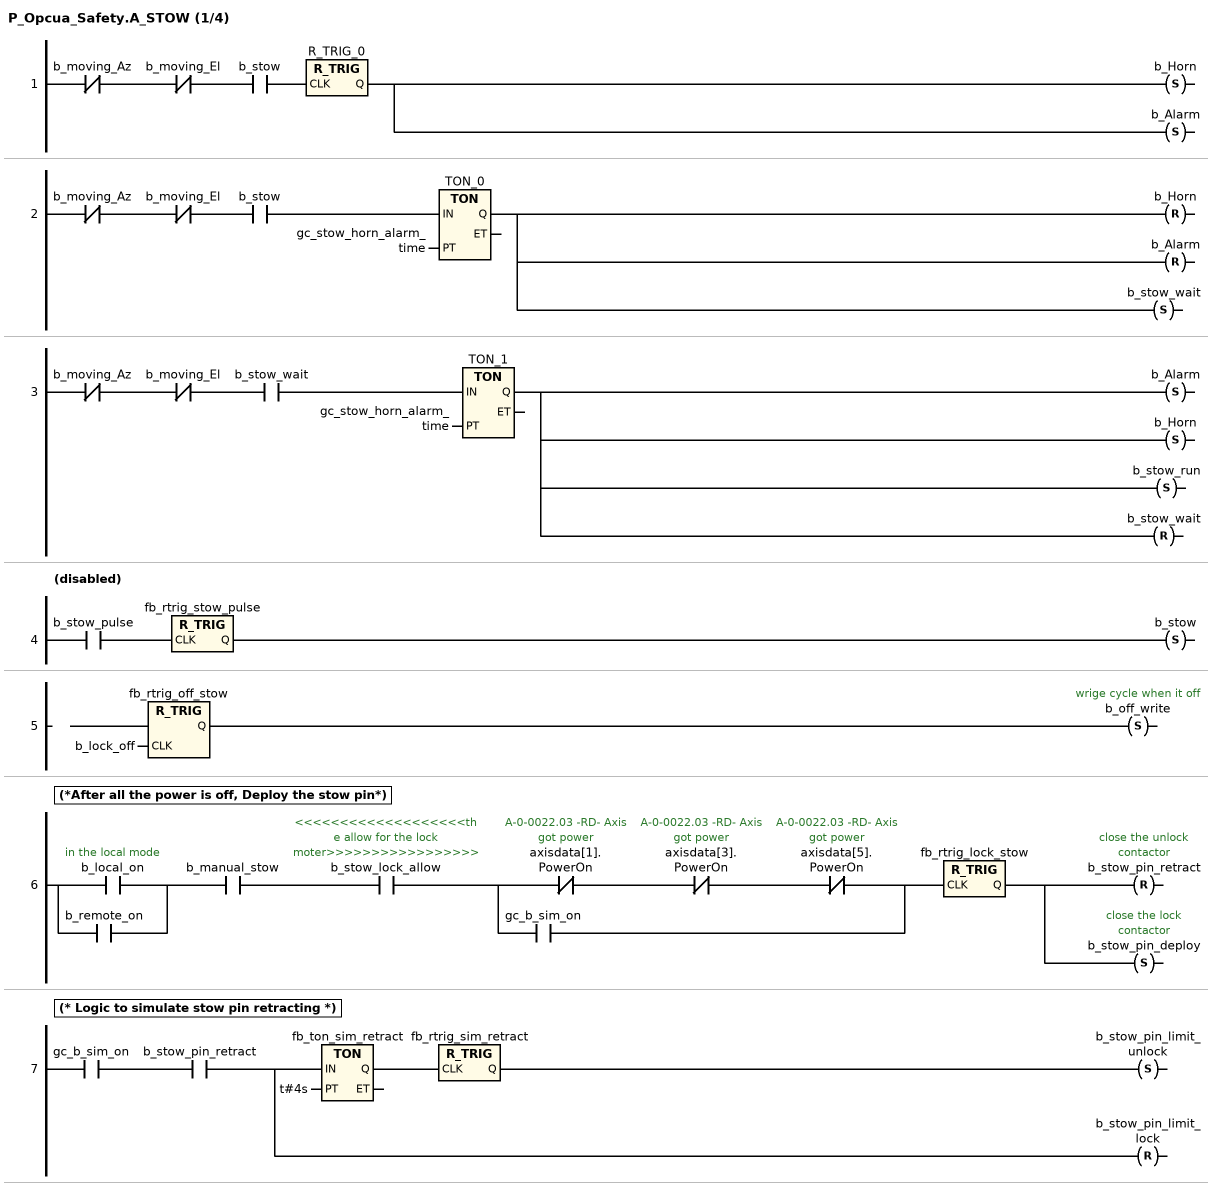
// NETWORK 1
R_TRIG_0(CLK := NOT b_moving_Az AND NOT b_moving_El AND b_stow); // R_TRIG
b_Horn S= R_TRIG_0.Q;
b_Alarm S= R_TRIG_0.Q;

// NETWORK 2
TON_0(IN := NOT b_moving_Az AND NOT b_moving_El AND b_stow, PT := gc_stow_horn_alarm_time); // TON
b_Horn R= TON_0.Q;
b_Alarm R= TON_0.Q;
b_stow_wait S= TON_0.Q;

// NETWORK 3
TON_1(IN := NOT b_moving_Az AND NOT b_moving_El AND b_stow_wait, PT := gc_stow_horn_alarm_time); // TON
b_Alarm S= TON_1.Q;
b_Horn S= TON_1.Q;
b_stow_run S= TON_1.Q;
b_stow_wait R= TON_1.Q;

// NETWORK 4 (disabled)
//   fb_rtrig_stow_pulse: the definition of rise trigger,The function block R_TRIG detects a rising edge.
// fb_rtrig_stow_pulse(CLK := b_stow_pulse); // R_TRIG
// b_stow S= fb_rtrig_stow_pulse.Q;

// NETWORK 5
//   b_lock_off: power off after arriving at the stow position
//   b_off_write: wrige cycle when it off
fb_rtrig_off_stow(CLK := b_lock_off); // R_TRIG
b_off_write S= fb_rtrig_off_stow.Q;

// NETWORK 6
//   fb_rtrig_lock_stow: the definition of rise trigger,The function block R_TRIG detects a rising edge.
//   b_local_on: in the local mode
//   b_stow_lock_allow: <<<<<<<<<<<<<<<<<<<the allow for the lock moter>>>>>>>>>>>>>>>>>
//   axisdata[1].PowerOn: A-0-0022.03 -RD- Axis got power
//   axisdata[3].PowerOn: A-0-0022.03 -RD- Axis got power
//   axisdata[5].PowerOn: A-0-0022.03 -RD- Axis got power
//   b_stow_pin_retract: close the unlock contactor
//   b_stow_pin_deploy: close the lock contactor
// label: (*After all the power is off, Deploy the stow pin*)
fb_rtrig_lock_stow(CLK := (b_local_on OR b_remote_on) AND b_manual_stow AND b_stow_lock_allow AND (NOT axisdata[1].PowerOn AND NOT axisdata[3].PowerOn AND NOT axisdata[5].PowerOn OR gc_b_sim_on)); // R_TRIG
b_stow_pin_retract R= fb_rtrig_lock_stow.Q;
b_stow_pin_deploy S= fb_rtrig_lock_stow.Q;

// NETWORK 7
//   fb_rtrig_sim_retract: the definition of rise trigger,The function block R_TRIG detects a rising edge.
//   fb_ton_sim_retract: The function block Timer On Delay implements a turn-on delay
// label: (* Logic to simulate stow pin retracting *)
_w1 := gc_b_sim_on AND b_stow_pin_retract;
fb_ton_sim_retract(IN := _w1, PT := t#4s); // TON
fb_rtrig_sim_retract(CLK := fb_ton_sim_retract.Q); // R_TRIG
b_stow_pin_limit_unlock S= fb_rtrig_sim_retract.Q;
b_stow_pin_limit_lock R= _w1;

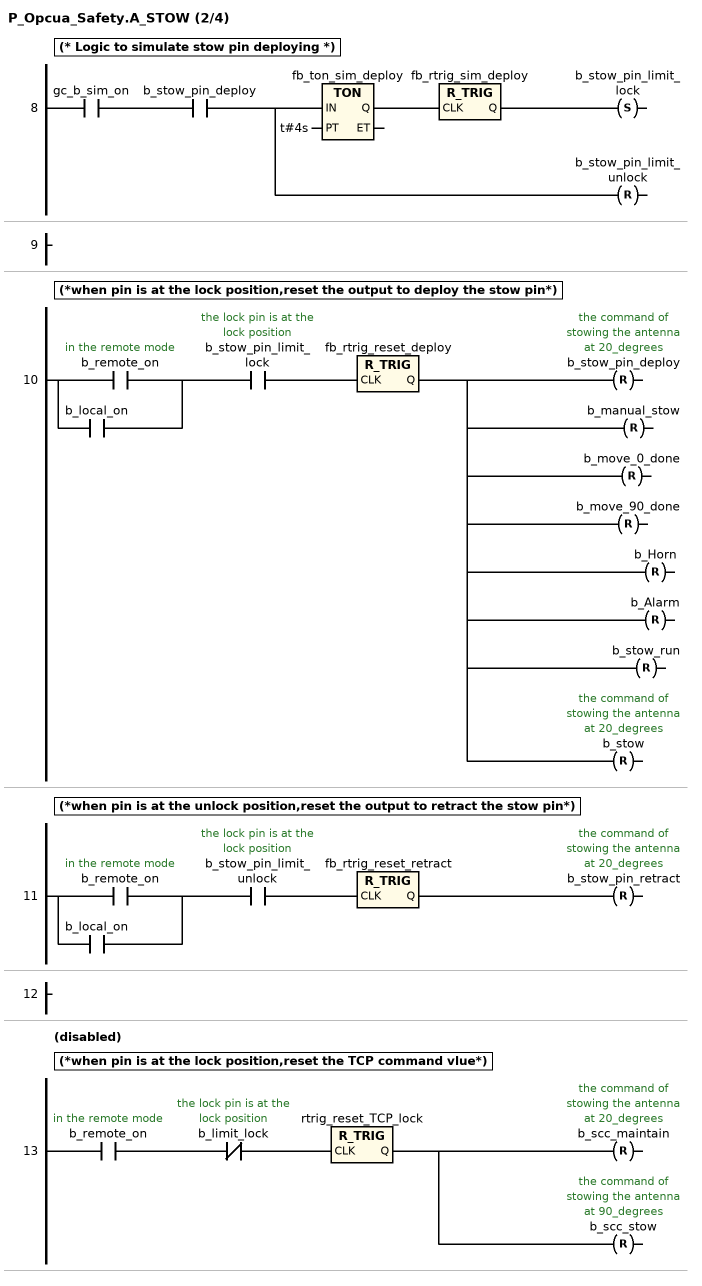
// NETWORK 8
//   fb_rtrig_sim_deploy: the definition of rise trigger,The function block R_TRIG detects a rising edge.
//   fb_ton_sim_deploy: The function block Timer On Delay implements a turn-on delay
// label: (* Logic to simulate stow pin deploying *)
_w2 := gc_b_sim_on AND b_stow_pin_deploy;
fb_ton_sim_deploy(IN := _w2, PT := t#4s); // TON
fb_rtrig_sim_deploy(CLK := fb_ton_sim_deploy.Q); // R_TRIG
b_stow_pin_limit_lock S= fb_rtrig_sim_deploy.Q;
b_stow_pin_limit_unlock R= _w2;

// NETWORK 9

// NETWORK 10
//   b_remote_on: in the remote mode
//   b_stow_pin_limit_lock: the lock pin is at the lock position
//   b_stow_pin_deploy: the command of stowing the antenna at 20_degrees
//   b_stow: the command of stowing the antenna at 20_degrees
// label: (*when pin is at the lock position,reset the output to deploy the stow pin*)
fb_rtrig_reset_deploy(CLK := (b_remote_on OR b_local_on) AND b_stow_pin_limit_lock); // R_TRIG
b_stow_pin_deploy R= fb_rtrig_reset_deploy.Q;
b_manual_stow R= fb_rtrig_reset_deploy.Q;
b_move_0_done R= fb_rtrig_reset_deploy.Q;
b_move_90_done R= fb_rtrig_reset_deploy.Q;
b_Horn R= fb_rtrig_reset_deploy.Q;
b_Alarm R= fb_rtrig_reset_deploy.Q;
b_stow_run R= fb_rtrig_reset_deploy.Q;
b_stow R= fb_rtrig_reset_deploy.Q;

// NETWORK 11
//   b_remote_on: in the remote mode
//   b_stow_pin_limit_unlock: the lock pin is at the lock position
//   b_stow_pin_retract: the command of stowing the antenna at 20_degrees
// label: (*when pin is at the unlock position,reset the output to retract the stow pin*)
fb_rtrig_reset_retract(CLK := (b_remote_on OR b_local_on) AND b_stow_pin_limit_unlock); // R_TRIG
b_stow_pin_retract R= fb_rtrig_reset_retract.Q;

// NETWORK 12

// NETWORK 13 (disabled)
//   b_remote_on: in the remote mode
//   b_limit_lock: the lock pin is at the lock position
//   b_scc_maintain: the command of stowing the antenna at 20_degrees
//   b_scc_stow: the command of stowing the antenna at 90_degrees
// label: (*when pin is at the lock position,reset the TCP command vlue*)
// rtrig_reset_TCP_lock(CLK := b_remote_on AND NOT b_limit_lock); // R_TRIG
// b_scc_maintain R= rtrig_reset_TCP_lock.Q;
// b_scc_stow R= rtrig_reset_TCP_lock.Q;

